LIN {X 0,Y 468.425,Z 168.39,A -85,B 0,C 180,E1 -7424.985,E2 -7424.985} C_VEL
LIN {X 0,Y 468.931,Z 154.374,A -85,B 0,C 180,E1 -7427.874,E2 -7427.874} C_VEL
LIN {X 0,Y 468.145,Z 148.139,A -85,B 0,C 180,E1 -7429.228,E2 -7429.228} C_VEL
LIN {X 0,Y 467.613,Z 145.238,A -85,B 0,C 180,E1 -7429.882,E2 -7429.882} C_VEL
LIN {X 0,Y 467.525,Z 145.248,A -85,B 0,C 180,E1 -7433.037,E2 -7433.037} C_VEL
LIN {X 0,Y 467.572,Z 145.242,A -85,B 0,C 180,E1 -7436.21,E2 -7436.21} C_VEL
LIN {X 0,Y 467.553,Z 145.24,A -85,B 0,C 180,E1 -7439.264,E2 -7439.264} C_VEL
LIN {X 0,Y 467.553,Z 145.247,A -85,B 0,C 180,E1 -7442.482,E2 -7442.482} C_VEL
LIN {X 0,Y 467.557,Z 145.24,A -85,B 0,C 180,E1 -7445.109,E2 -7445.109} C_VEL
LIN {X 0,Y 467.526,Z 145.247,A -85,B 0,C 180,E1 -7447.925,E2 -7447.925} C_VEL
LIN {X 0,Y 467.557,Z 145.242,A -85,B 0,C 180,E1 -7450.689,E2 -7450.689} C_VEL
LIN {X 0,Y 467.599,Z 145.243,A -85,B 0,C 180,E1 -7454.139,E2 -7454.139} C_VEL
LIN {X 0,Y 467.654,Z 145.23,A -85,B 0,C 180,E1 -7457.646,E2 -7457.646} C_VEL
LIN {X 0,Y 467.622,Z 145.234,A -85,B 0,C 180,E1 -7460.483,E2 -7460.483} C_VEL
LIN {X 0,Y 467.656,Z 145.227,A -85,B 0,C 180,E1 -7463.094,E2 -7463.094} C_VEL
LIN {X 0,Y 467.704,Z 145.221,A -85,B 0,C 180,E1 -7464.826,E2 -7464.826} C_VEL
LIN {X 0,Y 467.816,Z 145.21,A -85,B 0,C 180,E1 -7467.416,E2 -7467.416} C_VEL
LIN {X 0,Y 467.853,Z 145.208,A -85,B 0,C 180,E1 -7469.999,E2 -7469.999} C_VEL
LIN {X 0,Y 467.816,Z 145.207,A -85,B 0,C 180,E1 -7472.582,E2 -7472.582} C_VEL
LIN {X 0,Y 467.697,Z 145.226,A -85,B 0,C 180,E1 -7476.037,E2 -7476.037} C_VEL
LIN {X 0,Y 467.636,Z 145.23,A -85,B 0,C 180,E1 -7478.643,E2 -7478.643} C_VEL
LIN {X 0,Y 467.651,Z 145.228,A -85,B 0,C 180,E1 -7482.353,E2 -7482.353} C_VEL
LIN {X 0,Y 467.602,Z 145.237,A -85,B 0,C 180,E1 -7485.862,E2 -7485.862} C_VEL
LIN {X 0,Y 467.554,Z 145.247,A -85,B 0,C 180,E1 -7489.31,E2 -7489.31} C_VEL
LIN {X 0,Y 467.522,Z 145.244,A -85,B 0,C 180,E1 -7492.074,E2 -7492.074} C_VEL
LIN {X 0,Y 467.559,Z 145.242,A -85,B 0,C 180,E1 -7494.889,E2 -7494.889} C_VEL
LIN {X 0,Y 467.543,Z 145.243,A -85,B 0,C 180,E1 -7497.773,E2 -7497.773} C_VEL
LIN {X 0,Y 467.536,Z 145.249,A -85,B 0,C 180,E1 -7501.037,E2 -7501.037} C_VEL
LIN {X 0,Y 467.575,Z 145.237,A -85,B 0,C 180,E1 -7504.239,E2 -7504.239} C_VEL
LIN {X 0,Y 467.54,Z 145.248,A -85,B 0,C 180,E1 -7507.184,E2 -7507.184} C_VEL
LIN {X 0,Y 467.555,Z 145.24,A -85,B 0,C 180,E1 -7510.266,E2 -7510.266} C_VEL
LIN {X 0,Y 467.541,Z 145.242,A -85,B 0,C 180,E1 -7513.745,E2 -7513.745} C_VEL
LIN {X 0,Y 467.541,Z 145.243,A -85,B 0,C 180,E1 -7516.253,E2 -7516.253} C_VEL
LIN {X 0,Y 467.552,Z 145.24,A -85,B 0,C 180,E1 -7519.732,E2 -7519.732} C_VEL
LIN {X 0,Y 467.533,Z 145.249,A -85,B 0,C 180,E1 -7522.815,E2 -7522.815} C_VEL
LIN {X 0,Y 467.571,Z 145.238,A -85,B 0,C 180,E1 -7525.759,E2 -7525.759} C_VEL
LIN {X 0,Y 467.537,Z 145.245,A -85,B 0,C 180,E1 -7528.96,E2 -7528.96} C_VEL
LIN {X 0,Y 467.537,Z 145.246,A -85,B 0,C 180,E1 -7532.225,E2 -7532.225} C_VEL
LIN {X 0,Y 467.552,Z 145.241,A -85,B 0,C 180,E1 -7535.109,E2 -7535.109} C_VEL
LIN {X 0,Y 467.518,Z 145.247,A -85,B 0,C 180,E1 -7537.925,E2 -7537.925} C_VEL
LIN {X 0,Y 467.609,Z 145.237,A -85,B 0,C 180,E1 -7540.691,E2 -7540.691} C_VEL
LIN {X 0,Y 467.605,Z 145.241,A -85,B 0,C 180,E1 -7544.304,E2 -7544.304} C_VEL
LIN {X 0,Y 467.64,Z 145.233,A -85,B 0,C 180,E1 -7547.854,E2 -7547.854} C_VEL
LIN {X 0,Y 467.625,Z 145.231,A -85,B 0,C 180,E1 -7551.356,E2 -7551.356} C_VEL
LIN {X 0,Y 467.695,Z 145.229,A -85,B 0,C 180,E1 -7553.962,E2 -7553.962} C_VEL
LIN {X 0,Y 467.804,Z 145.21,A -85,B 0,C 180,E1 -7557.417,E2 -7557.417} C_VEL
LIN {X 0,Y 467.841,Z 145.212,A -85,B 0,C 180,E1 -7560,E2 -7560} C_VEL
LIN {X 0,Y 467.804,Z 145.209,A -85,B 0,C 180,E1 -7562.583,E2 -7562.583} C_VEL
LIN {X 0,Y 467.692,Z 145.228,A -85,B 0,C 180,E1 -7566.038,E2 -7566.038} C_VEL
LIN {X 0,Y 467.624,Z 145.231,A -85,B 0,C 180,E1 -7568.644,E2 -7568.644} C_VEL
LIN {X 0,Y 467.639,Z 145.232,A -85,B 0,C 180,E1 -7572.146,E2 -7572.146} C_VEL
LIN {X 0,Y 467.604,Z 145.241,A -85,B 0,C 180,E1 -7575.696,E2 -7575.696} C_VEL
LIN {X 0,Y 467.564,Z 145.239,A -85,B 0,C 180,E1 -7578.748,E2 -7578.748} C_VEL
LIN {X 0,Y 467.55,Z 145.245,A -85,B 0,C 180,E1 -7581.261,E2 -7581.261} C_VEL
LIN {X 0,Y 467.541,Z 145.244,A -85,B 0,C 180,E1 -7583.945,E2 -7583.945} C_VEL
LIN {X 0,Y 467.526,Z 145.245,A -85,B 0,C 180,E1 -7586.806,E2 -7586.806} C_VEL
LIN {X 0,Y 467.502,Z 145.249,A -85,B 0,C 180,E1 -7589.742,E2 -7589.742} C_VEL
LIN {X 0,Y 467.565,Z 145.241,A -85,B 0,C 180,E1 -7592.76,E2 -7592.76} C_VEL
LIN {X 0,Y 467.536,Z 145.243,A -85,B 0,C 180,E1 -7595.891,E2 -7595.891} C_VEL
LIN {X 0,Y 467.536,Z 145.25,A -85,B 0,C 180,E1 -7599.149,E2 -7599.149} C_VEL
LIN {X 0,Y 467.552,Z 145.244,A -85,B 0,C 180,E1 -7601.406,E2 -7601.406} C_VEL
LIN {X 0,Y 467.556,Z 145.247,A -85,B 0,C 180,E1 -7605.053,E2 -7605.053} C_VEL
LIN {X 0,Y 467.555,Z 145.245,A -85,B 0,C 180,E1 -7608.727,E2 -7608.727} C_VEL
LIN {X 0,Y 467.535,Z 145.242,A -85,B 0,C 180,E1 -7611.954,E2 -7611.954} C_VEL
LIN {X 0,Y 467.545,Z 145.244,A -85,B 0,C 180,E1 -7615.167,E2 -7615.167} C_VEL
LIN {X 0,Y 467.542,Z 145.244,A -85,B 0,C 180,E1 -7618.258,E2 -7618.258} C_VEL
LIN {X 0,Y 467.521,Z 145.247,A -85,B 0,C 180,E1 -7621.248,E2 -7621.248} C_VEL
LIN {X 0,Y 467.555,Z 145.345,A -85,B 0,C 180,E1 -7624.376,E2 -7624.376} C_VEL
LIN {X 0,Y 469.577,Z 155.706,A -85,B 0,C 180,E1 -7626.4,E2 -7626.4} C_VEL
LIN {X 0,Y 469.686,Z 160.79,A -85,B 0,C 180,E1 -7627.338,E2 -7627.338} C_VEL
LIN {X 0,Y 469.023,Z 174.71,A -85,B 0,C 180,E1 -7629.841,E2 -7629.841} C_VEL
LIN {X 0,Y 468.327,Z 192.765,A -85,B 0,C 180,E1 -7633.041,E2 -7633.041} C_VEL
LIN {X 0,Y 471.066,Z 211.841,A -85,B 0,C 180,E1 -7633.457,E2 -7633.457} C_VEL
LIN {X 0,Y 470.265,Z 300.839,A -85,B 0,C 180,E1 -7634.923,E2 -7634.923} C_VEL
LIN {X 0,Y 469.84,Z 314.649,A -85,B 0,C 180,E1 -7635.325,E2 -7635.325} C_VEL
LIN {X 0,Y 469.462,Z 327.139,A -85,B 0,C 180,E1 -7635.866,E2 -7635.866} C_VEL
LIN {X 0,Y 468.985,Z 339.105,A -85,B 0,C 180,E1 -7636.57,E2 -7636.57} C_VEL
LIN {X 0,Y 468.506,Z 350.327,A -85,B 0,C 180,E1 -7637.415,E2 -7637.415} C_VEL
LIN {X 0,Y 468.06,Z 360.974,A -85,B 0,C 180,E1 -7638.415,E2 -7638.415} C_VEL
LIN {X 0,Y 467.63,Z 369.45,A -85,B 0,C 180,E1 -7639.392,E2 -7639.392} C_VEL
LIN {X 0,Y 467.262,Z 378.639,A -85,B 0,C 180,E1 -7640.696,E2 -7640.696} C_VEL
LIN {X 0,Y 467.005,Z 386.039,A -85,B 0,C 180,E1 -7641.999,E2 -7641.999} C_VEL
LIN {X 0,Y 466.832,Z 391.044,A -85,B 0,C 180,E1 -7643.083,E2 -7643.083} C_VEL
LIN {X 0,Y 466.755,Z 395.897,A -85,B 0,C 180,E1 -7644.384,E2 -7644.384} C_VEL
LIN {X 0,Y 466.645,Z 399.603,A -85,B 0,C 180,E1 -7645.682,E2 -7645.682} C_VEL
LIN {X 0,Y 466.688,Z 401.518,A -85,B 0,C 180,E1 -7646.547,E2 -7646.547} C_VEL
LIN {X 0,Y 466.662,Z 402.961,A -85,B 0,C 180,E1 -7647.411,E2 -7647.411} C_VEL
LIN {X 0,Y 466.62,Z 404.599,A -85,B 0,C 180,E1 -7649.138,E2 -7649.138} C_VEL
LIN {X 0,Y 466.601,Z 404.823,A -85,B 0,C 180,E1 -7650.001,E2 -7650.001} C_VEL
LIN {X 0,Y 466.62,Z 404.604,A -85,B 0,C 180,E1 -7650.864,E2 -7650.864} C_VEL
LIN {X 0,Y 466.662,Z 402.957,A -85,B 0,C 180,E1 -7652.59,E2 -7652.59} C_VEL
LIN {X 0,Y 466.688,Z 401.525,A -85,B 0,C 180,E1 -7653.454,E2 -7653.454} C_VEL
LIN {X 0,Y 466.687,Z 398.517,A -85,B 0,C 180,E1 -7654.752,E2 -7654.752} C_VEL
LIN {X 0,Y 466.743,Z 394.447,A -85,B 0,C 180,E1 -7656.051,E2 -7656.051} C_VEL
LIN {X 0,Y 466.94,Z 388.181,A -85,B 0,C 180,E1 -7657.568,E2 -7657.568} C_VEL
LIN {X 0,Y 467.178,Z 381.351,A -85,B 0,C 180,E1 -7658.871,E2 -7658.871} C_VEL
LIN {X 0,Y 467.489,Z 372.873,A -85,B 0,C 180,E1 -7660.175,E2 -7660.175} C_VEL
LIN {X 0,Y 467.968,Z 364.14,A -85,B 0,C 180,E1 -7661.259,E2 -7661.259} C_VEL
LIN {X 0,Y 468.42,Z 354.024,A -85,B 0,C 180,E1 -7662.287,E2 -7662.287} C_VEL
LIN {X 0,Y 468.849,Z 342.723,A -85,B 0,C 180,E1 -7663.215,E2 -7663.215} C_VEL
LIN {X 0,Y 469.375,Z 330.864,A -85,B 0,C 180,E1 -7663.972,E2 -7663.972} C_VEL
LIN {X 0,Y 469.874,Z 317.322,A -85,B 0,C 180,E1 -7664.62,E2 -7664.62} C_VEL
LIN {X 0,Y 470.259,Z 305.288,A -85,B 0,C 180,E1 -7665.023,E2 -7665.023} C_VEL
LIN {X 0,Y 470.505,Z 290.619,A -85,B 0,C 180,E1 -7665.32,E2 -7665.32} C_VEL
LIN {X 0,Y 471.152,Z 209.638,A -85,B 0,C 180,E1 -7666.67,E2 -7666.67} C_VEL
LIN {X 0,Y 468.296,Z 191.81,A -85,B 0,C 180,E1 -7667.102,E2 -7667.102} C_VEL
LIN {X 0,Y 468.849,Z 176.842,A -85,B 0,C 180,E1 -7669.711,E2 -7669.711} C_VEL
LIN {X 0,Y 469.422,Z 162.683,A -85,B 0,C 180,E1 -7672.213,E2 -7672.213} C_VEL
LIN {X 0,Y 469.596,Z 156.216,A -85,B 0,C 180,E1 -7673.366,E2 -7673.366} C_VEL
LIN {X 0,Y 467.567,Z 145.248,A -85,B 0,C 180,E1 -7675.477,E2 -7675.477} C_VEL
LIN {X 0,Y 467.527,Z 145.25,A -85,B 0,C 180,E1 -7678.754,E2 -7678.754} C_VEL
LIN {X 0,Y 467.549,Z 145.246,A -85,B 0,C 180,E1 -7681.743,E2 -7681.743} C_VEL
LIN {X 0,Y 467.553,Z 145.246,A -85,B 0,C 180,E1 -7684.834,E2 -7684.834} C_VEL
LIN {X 0,Y 467.543,Z 145.243,A -85,B 0,C 180,E1 -7688.047,E2 -7688.047} C_VEL
LIN {X 0,Y 467.563,Z 145.243,A -85,B 0,C 180,E1 -7691.275,E2 -7691.275} C_VEL
LIN {X 0,Y 467.568,Z 145.243,A -85,B 0,C 180,E1 -7694.948,E2 -7694.948} C_VEL
LIN {X 0,Y 467.561,Z 145.242,A -85,B 0,C 180,E1 -7698.595,E2 -7698.595} C_VEL
LIN {X 0,Y 467.546,Z 145.24,A -85,B 0,C 180,E1 -7701.412,E2 -7701.412} C_VEL
LIN {X 0,Y 467.558,Z 145.242,A -85,B 0,C 180,E1 -7704.262,E2 -7704.262} C_VEL
LIN {X 0,Y 467.576,Z 145.239,A -85,B 0,C 180,E1 -7707.323,E2 -7707.323} C_VEL
LIN {X 0,Y 467.548,Z 145.245,A -85,B 0,C 180,E1 -7710.673,E2 -7710.673} C_VEL
LIN {X 0,Y 467.537,Z 145.243,A -85,B 0,C 180,E1 -7713.195,E2 -7713.195} C_VEL
LIN {X 0,Y 467.559,Z 145.245,A -85,B 0,C 180,E1 -7716.056,E2 -7716.056} C_VEL
LIN {X 0,Y 467.622,Z 145.233,A -85,B 0,C 180,E1 -7719.777,E2 -7719.777} C_VEL
LIN {X 0,Y 467.569,Z 145.243,A -85,B 0,C 180,E1 -7722.505,E2 -7722.505} C_VEL
LIN {X 0,Y 467.598,Z 145.237,A -85,B 0,C 180,E1 -7725.196,E2 -7725.196} C_VEL
LIN {X 0,Y 467.66,Z 145.234,A -85,B 0,C 180,E1 -7727.855,E2 -7727.855} C_VEL
LIN {X 0,Y 467.661,Z 145.232,A -85,B 0,C 180,E1 -7731.357,E2 -7731.357} C_VEL
LIN {X 0,Y 467.706,Z 145.23,A -85,B 0,C 180,E1 -7733.962,E2 -7733.962} C_VEL
LIN {X 0,Y 467.818,Z 145.214,A -85,B 0,C 180,E1 -7737.417,E2 -7737.417} C_VEL
LIN {X 0,Y 467.856,Z 145.211,A -85,B 0,C 180,E1 -7740,E2 -7740} C_VEL
LIN {X 0,Y 467.853,Z 145.209,A -85,B 0,C 180,E1 -7742.583,E2 -7742.583} C_VEL
LIN {X 0,Y 467.724,Z 145.348,A -85,B 0,C 180,E1 -7746.444,E2 -7746.444} C_VEL
LIN {X 0,Y 468.878,Z 151.823,A -85,B 0,C 180,E1 -7747.753,E2 -7747.753} C_VEL
LIN {X 0,Y 468.773,Z 162.022,A -85,B 0,C 180,E1 -7749.71,E2 -7749.71} C_VEL
LIN {X 0,Y 468.622,Z 168.72,A -85,B 0,C 180,E1 -7750.969,E2 -7750.969} C_VEL
LIN {X 0,Y 471.42,Z 183.099,A -85,B 0,C 180,E1 -7751.339,E2 -7751.339} C_VEL
LIN {X 0,Y 470.458,Z 276.646,A -85,B 0,C 180,E1 -7752.922,E2 -7752.922} C_VEL
LIN {X 0,Y 470.148,Z 290.015,A -85,B 0,C 180,E1 -7753.322,E2 -7753.322} C_VEL
LIN {X 0,Y 469.795,Z 303.075,A -85,B 0,C 180,E1 -7753.904,E2 -7753.904} C_VEL
LIN {X 0,Y 469.333,Z 315.18,A -85,B 0,C 180,E1 -7754.637,E2 -7754.637} C_VEL
LIN {X 0,Y 468.823,Z 326.843,A -85,B 0,C 180,E1 -7755.543,E2 -7755.543} C_VEL
LIN {X 0,Y 468.316,Z 337.266,A -85,B 0,C 180,E1 -7756.567,E2 -7756.567} C_VEL
LIN {X 0,Y 467.878,Z 346.668,A -85,B 0,C 180,E1 -7757.709,E2 -7757.709} C_VEL
LIN {X 0,Y 467.493,Z 355.126,A -85,B 0,C 180,E1 -7758.975,E2 -7758.975} C_VEL
LIN {X 0,Y 467.146,Z 361.925,A -85,B 0,C 180,E1 -7760.245,E2 -7760.245} C_VEL
LIN {X 0,Y 466.949,Z 367.849,A -85,B 0,C 180,E1 -7761.639,E2 -7761.639} C_VEL
LIN {X 0,Y 466.798,Z 372.451,A -85,B 0,C 180,E1 -7763.045,E2 -7763.045} C_VEL
LIN {X 0,Y 466.725,Z 374.852,A -85,B 0,C 180,E1 -7763.99,E2 -7763.99} C_VEL
LIN {X 0,Y 466.556,Z 377.331,A -85,B 0,C 180,E1 -7765.335,E2 -7765.335} C_VEL
LIN {X 0,Y 466.544,Z 378.893,A -85,B 0,C 180,E1 -7766.867,E2 -7766.867} C_VEL
LIN {X 0,Y 466.505,Z 379.236,A -85,B 0,C 180,E1 -7767.842,E2 -7767.842} C_VEL
LIN {X 0,Y 466.532,Z 378.9,A -85,B 0,C 180,E1 -7769.104,E2 -7769.104} C_VEL
LIN {X 0,Y 466.628,Z 377.107,A -85,B 0,C 180,E1 -7770.803,E2 -7770.803} C_VEL
LIN {X 0,Y 466.699,Z 375.248,A -85,B 0,C 180,E1 -7771.808,E2 -7771.808} C_VEL
LIN {X 0,Y 466.779,Z 371.323,A -85,B 0,C 180,E1 -7773.337,E2 -7773.337} C_VEL
LIN {X 0,Y 466.91,Z 367.439,A -85,B 0,C 180,E1 -7774.463,E2 -7774.463} C_VEL
LIN {X 0,Y 467.154,Z 361.069,A -85,B 0,C 180,E1 -7775.926,E2 -7775.926} C_VEL
LIN {X 0,Y 467.5,Z 353.312,A -85,B 0,C 180,E1 -7777.309,E2 -7777.309} C_VEL
LIN {X 0,Y 467.913,Z 343.957,A -85,B 0,C 180,E1 -7778.644,E2 -7778.644} C_VEL
LIN {X 0,Y 468.329,Z 334.292,A -85,B 0,C 180,E1 -7779.744,E2 -7779.744} C_VEL
LIN {X 0,Y 468.739,Z 323.844,A -85,B 0,C 180,E1 -7780.709,E2 -7780.709} C_VEL
LIN {X 0,Y 469.264,Z 311.997,A -85,B 0,C 180,E1 -7781.579,E2 -7781.579} C_VEL
LIN {X 0,Y 469.719,Z 299.794,A -85,B 0,C 180,E1 -7782.263,E2 -7782.263} C_VEL
LIN {X 0,Y 470.054,Z 286.143,A -85,B 0,C 180,E1 -7782.823,E2 -7782.823} C_VEL
LIN {X 0,Y 470.329,Z 272.94,A -85,B 0,C 180,E1 -7783.165,E2 -7783.165} C_VEL
LIN {X 0,Y 470.929,Z 213.093,A -85,B 0,C 180,E1 -7784.14,E2 -7784.14} C_VEL
LIN {X 0,Y 470.465,Z 207.289,A -85,B 0,C 180,E1 -7784.254,E2 -7784.254} C_VEL
LIN {X 0,Y 468.205,Z 197.882,A -85,B 0,C 180,E1 -7784.487,E2 -7784.487} C_VEL
LIN {X 0,Y 465.943,Z 190.424,A -85,B 0,C 180,E1 -7784.691,E2 -7784.691} C_VEL
LIN {X 0,Y 464.135,Z 182.84,A -85,B 0,C 180,E1 -7784.882,E2 -7784.882} C_VEL
LIN {X 0,Y 461.432,Z 168.53,A -85,B 0,C 180,E1 -7785.235,E2 -7785.235} C_VEL
LIN {X 0,Y 461.964,Z 155.386,A -85,B 0,C 180,E1 -7787.98,E2 -7787.98} C_VEL
LIN {X 0,Y 461.065,Z 148.726,A -85,B 0,C 180,E1 -7789.445,E2 -7789.445} C_VEL
LIN {X 0,Y 460.572,Z 146.116,A -85,B 0,C 180,E1 -7790.053,E2 -7790.053} C_VEL
LIN {X 0,Y 460.475,Z 146.124,A -85,B 0,C 180,E1 -7793.47,E2 -7793.47} C_VEL
LIN {X 0,Y 460.522,Z 146.122,A -85,B 0,C 180,E1 -7796.674,E2 -7796.674} C_VEL
LIN {X 0,Y 460.49,Z 146.121,A -85,B 0,C 180,E1 -7799.758,E2 -7799.758} C_VEL
LIN {X 0,Y 460.493,Z 146.123,A -85,B 0,C 180,E1 -7802.75,E2 -7802.75} C_VEL
LIN {X 0,Y 460.517,Z 146.117,A -85,B 0,C 180,E1 -7805.666,E2 -7805.666} C_VEL
LIN {X 0,Y 460.519,Z 146.12,A -85,B 0,C 180,E1 -7808.581,E2 -7808.581} C_VEL
LIN {X 0,Y 460.535,Z 146.114,A -85,B 0,C 180,E1 -7811.308,E2 -7811.308} C_VEL
LIN {X 0,Y 460.572,Z 146.117,A -85,B 0,C 180,E1 -7814.057,E2 -7814.057} C_VEL
LIN {X 0,Y 460.609,Z 146.108,A -85,B 0,C 180,E1 -7817.665,E2 -7817.665} C_VEL
LIN {X 0,Y 460.593,Z 146.107,A -85,B 0,C 180,E1 -7821.222,E2 -7821.222} C_VEL
LIN {X 0,Y 460.672,Z 146.105,A -85,B 0,C 180,E1 -7823.869,E2 -7823.869} C_VEL
LIN {X 0,Y 460.759,Z 146.088,A -85,B 0,C 180,E1 -7827.377,E2 -7827.377} C_VEL
LIN {X 0,Y 460.823,Z 146.084,A -85,B 0,C 180,E1 -7829.999,E2 -7829.999} C_VEL
LIN {X 0,Y 460.759,Z 146.086,A -85,B 0,C 180,E1 -7832.622,E2 -7832.622} C_VEL
LIN {X 0,Y 460.664,Z 146.101,A -85,B 0,C 180,E1 -7836.13,E2 -7836.13} C_VEL
LIN {X 0,Y 460.591,Z 146.107,A -85,B 0,C 180,E1 -7838.776,E2 -7838.776} C_VEL
LIN {X 0,Y 460.6,Z 146.106,A -85,B 0,C 180,E1 -7842.434,E2 -7842.434} C_VEL
LIN {X 0,Y 460.559,Z 146.113,A -85,B 0,C 180,E1 -7845.977,E2 -7845.977} C_VEL
LIN {X 0,Y 460.532,Z 146.116,A -85,B 0,C 180,E1 -7848.885,E2 -7848.885} C_VEL
LIN {X 0,Y 460.51,Z 146.124,A -85,B 0,C 180,E1 -7851.485,E2 -7851.485} C_VEL
LIN {X 0,Y 460.517,Z 146.116,A -85,B 0,C 180,E1 -7854.333,E2 -7854.333} C_VEL
LIN {X 0,Y 460.491,Z 146.128,A -85,B 0,C 180,E1 -7857.248,E2 -7857.248} C_VEL
LIN {X 0,Y 460.493,Z 146.12,A -85,B 0,C 180,E1 -7860.24,E2 -7860.24} C_VEL
LIN {X 0,Y 460.515,Z 146.122,A -85,B 0,C 180,E1 -7863.325,E2 -7863.325} C_VEL
LIN {X 0,Y 460.47,Z 146.124,A -85,B 0,C 180,E1 -7866.529,E2 -7866.529} C_VEL
LIN {X 0,Y 460.51,Z 146.117,A -85,B 0,C 180,E1 -7869.863,E2 -7869.863} C_VEL
LIN {X 0,Y 460.459,Z 146.132,A -85,B 0,C 180,E1 -7872.892,E2 -7872.892} C_VEL
LIN {X 0,Y 460.499,Z 146.119,A -85,B 0,C 180,E1 -7875.831,E2 -7875.831} C_VEL
LIN {X 0,Y 460.51,Z 146.123,A -85,B 0,C 180,E1 -7878.986,E2 -7878.986} C_VEL
LIN {X 0,Y 460.489,Z 146.124,A -85,B 0,C 180,E1 -7882.375,E2 -7882.375} C_VEL
LIN {X 0,Y 460.53,Z 146.115,A -85,B 0,C 180,E1 -7885.622,E2 -7885.622} C_VEL
LIN {X 0,Y 460.498,Z 146.125,A -85,B 0,C 180,E1 -7888.741,E2 -7888.741} C_VEL
LIN {X 0,Y 460.498,Z 146.119,A -85,B 0,C 180,E1 -7891.763,E2 -7891.763} C_VEL
LIN {X 0,Y 460.516,Z 146.122,A -85,B 0,C 180,E1 -7894.702,E2 -7894.702} C_VEL
LIN {X 0,Y 460.496,Z 146.119,A -85,B 0,C 180,E1 -7897.57,E2 -7897.57} C_VEL
LIN {X 0,Y 460.554,Z 146.12,A -85,B 0,C 180,E1 -7900.384,E2 -7900.384} C_VEL
LIN {X 0,Y 460.56,Z 146.116,A -85,B 0,C 180,E1 -7904.057,E2 -7904.057} C_VEL
LIN {X 0,Y 460.596,Z 146.108,A -85,B 0,C 180,E1 -7907.665,E2 -7907.665} C_VEL
LIN {X 0,Y 460.58,Z 146.109,A -85,B 0,C 180,E1 -7911.223,E2 -7911.223} C_VEL
LIN {X 0,Y 460.661,Z 146.104,A -85,B 0,C 180,E1 -7913.869,E2 -7913.869} C_VEL
LIN {X 0,Y 460.748,Z 146.089,A -85,B 0,C 180,E1 -7917.377,E2 -7917.377} C_VEL
LIN {X 0,Y 460.811,Z 146.087,A -85,B 0,C 180,E1 -7920,E2 -7920} C_VEL
LIN {X 0,Y 460.747,Z 146.088,A -85,B 0,C 180,E1 -7922.623,E2 -7922.623} C_VEL
LIN {X 0,Y 460.658,Z 146.103,A -85,B 0,C 180,E1 -7926.13,E2 -7926.13} C_VEL
LIN {X 0,Y 460.579,Z 146.109,A -85,B 0,C 180,E1 -7928.777,E2 -7928.777} C_VEL
LIN {X 0,Y 460.589,Z 146.108,A -85,B 0,C 180,E1 -7932.435,E2 -7932.435} C_VEL
LIN {X 0,Y 460.549,Z 146.116,A -85,B 0,C 180,E1 -7935.978,E2 -7935.978} C_VEL
LIN {X 0,Y 460.522,Z 146.117,A -85,B 0,C 180,E1 -7938.887,E2 -7938.887} C_VEL
LIN {X 0,Y 460.501,Z 146.127,A -85,B 0,C 180,E1 -7941.486,E2 -7941.486} C_VEL
LIN {X 0,Y 460.505,Z 146.118,A -85,B 0,C 180,E1 -7944.334,E2 -7944.334} C_VEL
LIN {X 0,Y 460.481,Z 146.127,A -85,B 0,C 180,E1 -7947.25,E2 -7947.25} C_VEL
LIN {X 0,Y 460.471,Z 146.122,A -85,B 0,C 180,E1 -7950.243,E2 -7950.243} C_VEL
LIN {X 0,Y 460.508,Z 146.125,A -85,B 0,C 180,E1 -7953.327,E2 -7953.327} C_VEL
LIN {X 0,Y 460.453,Z 146.125,A -85,B 0,C 180,E1 -7956.532,E2 -7956.532} C_VEL
LIN {X 0,Y 460.503,Z 146.119,A -85,B 0,C 180,E1 -7959.865,E2 -7959.865} C_VEL
LIN {X 0,Y 460.45,Z 146.131,A -85,B 0,C 180,E1 -7962.893,E2 -7962.893} C_VEL
LIN {X 0,Y 460.498,Z 146.119,A -85,B 0,C 180,E1 -7965.832,E2 -7965.832} C_VEL
LIN {X 0,Y 460.509,Z 146.125,A -85,B 0,C 180,E1 -7968.988,E2 -7968.988} C_VEL
LIN {X 0,Y 460.478,Z 146.124,A -85,B 0,C 180,E1 -7972.376,E2 -7972.376} C_VEL
LIN {X 0,Y 460.529,Z 146.115,A -85,B 0,C 180,E1 -7975.623,E2 -7975.623} C_VEL
LIN {X 0,Y 460.501,Z 146.127,A -85,B 0,C 180,E1 -7978.743,E2 -7978.743} C_VEL
LIN {X 0,Y 460.493,Z 146.121,A -85,B 0,C 180,E1 -7981.764,E2 -7981.764} C_VEL
LIN {X 0,Y 460.544,Z 146.127,A -85,B 0,C 180,E1 -7984.16,E2 -7984.16} C_VEL
LIN {X 0,Y 462.734,Z 157.978,A -85,B 0,C 180,E1 -7986.505,E2 -7986.505} C_VEL
LIN {X 0,Y 462.406,Z 169.387,A -85,B 0,C 180,E1 -7988.607,E2 -7988.607} C_VEL
LIN {X 0,Y 461.565,Z 185.829,A -85,B 0,C 180,E1 -7991.583,E2 -7991.583} C_VEL
LIN {X 0,Y 461.332,Z 192.537,A -85,B 0,C 180,E1 -7992.79,E2 -7992.79} C_VEL
LIN {X 0,Y 464.237,Z 212.61,A -85,B 0,C 180,E1 -7993.238,E2 -7993.238} C_VEL
LIN {X 0,Y 463.352,Z 301.882,A -85,B 0,C 180,E1 -7994.749,E2 -7994.749} C_VEL
LIN {X 0,Y 462.91,Z 315.28,A -85,B 0,C 180,E1 -7995.156,E2 -7995.156} C_VEL
LIN {X 0,Y 462.495,Z 327.522,A -85,B 0,C 180,E1 -7995.705,E2 -7995.705} C_VEL
LIN {X 0,Y 461.97,Z 340.146,A -85,B 0,C 180,E1 -7996.474,E2 -7996.474} C_VEL
LIN {X 0,Y 461.451,Z 351.822,A -85,B 0,C 180,E1 -7997.389,E2 -7997.389} C_VEL
LIN {X 0,Y 461.005,Z 361.575,A -85,B 0,C 180,E1 -7998.347,E2 -7998.347} C_VEL
LIN {X 0,Y 460.515,Z 370.744,A -85,B 0,C 180,E1 -7999.448,E2 -7999.448} C_VEL
LIN {X 0,Y 460.173,Z 379.692,A -85,B 0,C 180,E1 -8000.773,E2 -8000.773} C_VEL
LIN {X 0,Y 459.887,Z 386.845,A -85,B 0,C 180,E1 -8002.095,E2 -8002.095} C_VEL
LIN {X 0,Y 459.713,Z 393.112,A -85,B 0,C 180,E1 -8003.57,E2 -8003.57} C_VEL
LIN {X 0,Y 459.614,Z 398.275,A -85,B 0,C 180,E1 -8005.176,E2 -8005.176} C_VEL
LIN {X 0,Y 459.583,Z 401.294,A -85,B 0,C 180,E1 -8006.494,E2 -8006.494} C_VEL
LIN {X 0,Y 459.584,Z 402.749,A -85,B 0,C 180,E1 -8007.371,E2 -8007.371} C_VEL
LIN {X 0,Y 459.523,Z 404.397,A -85,B 0,C 180,E1 -8009.124,E2 -8009.124} C_VEL
LIN {X 0,Y 459.532,Z 404.627,A -85,B 0,C 180,E1 -8010.001,E2 -8010.001} C_VEL
LIN {X 0,Y 459.523,Z 404.413,A -85,B 0,C 180,E1 -8010.877,E2 -8010.877} C_VEL
LIN {X 0,Y 459.584,Z 402.77,A -85,B 0,C 180,E1 -8012.63,E2 -8012.63} C_VEL
LIN {X 0,Y 459.583,Z 401.339,A -85,B 0,C 180,E1 -8013.508,E2 -8013.508} C_VEL
LIN {X 0,Y 459.615,Z 398.334,A -85,B 0,C 180,E1 -8014.825,E2 -8014.825} C_VEL
LIN {X 0,Y 459.693,Z 393.3,A -85,B 0,C 180,E1 -8016.407,E2 -8016.407} C_VEL
LIN {X 0,Y 459.891,Z 386.977,A -85,B 0,C 180,E1 -8017.906,E2 -8017.906} C_VEL
LIN {X 0,Y 460.177,Z 379.912,A -85,B 0,C 180,E1 -8019.229,E2 -8019.229} C_VEL
LIN {X 0,Y 460.534,Z 371.052,A -85,B 0,C 180,E1 -8020.553,E2 -8020.553} C_VEL
LIN {X 0,Y 461.1,Z 361.007,A -85,B 0,C 180,E1 -8021.763,E2 -8021.763} C_VEL
LIN {X 0,Y 461.561,Z 350.198,A -85,B 0,C 180,E1 -8022.807,E2 -8022.807} C_VEL
LIN {X 0,Y 462.082,Z 339.476,A -85,B 0,C 180,E1 -8023.636,E2 -8023.636} C_VEL
LIN {X 0,Y 462.65,Z 326.791,A -85,B 0,C 180,E1 -8024.404,E2 -8024.404} C_VEL
LIN {X 0,Y 463.144,Z 313.719,A -85,B 0,C 180,E1 -8024.978,E2 -8024.978} C_VEL
LIN {X 0,Y 463.549,Z 300.995,A -85,B 0,C 180,E1 -8025.359,E2 -8025.359} C_VEL
LIN {X 0,Y 464.427,Z 210.669,A -85,B 0,C 180,E1 -8026.92,E2 -8026.92} C_VEL
LIN {X 0,Y 461.386,Z 191.495,A -85,B 0,C 180,E1 -8027.407,E2 -8027.407} C_VEL
LIN {X 0,Y 461.973,Z 175.505,A -85,B 0,C 180,E1 -8030.249,E2 -8030.249} C_VEL
LIN {X 0,Y 462.713,Z 160.018,A -85,B 0,C 180,E1 -8033.024,E2 -8033.024} C_VEL
LIN {X 0,Y 462.253,Z 154.911,A -85,B 0,C 180,E1 -8033.989,E2 -8033.989} C_VEL
LIN {X 0,Y 460.533,Z 146.124,A -85,B 0,C 180,E1 -8035.736,E2 -8035.736} C_VEL
LIN {X 0,Y 460.498,Z 146.124,A -85,B 0,C 180,E1 -8038.237,E2 -8038.237} C_VEL
LIN {X 0,Y 460.498,Z 146.126,A -85,B 0,C 180,E1 -8041.278,E2 -8041.278} C_VEL
LIN {X 0,Y 460.522,Z 146.119,A -85,B 0,C 180,E1 -8044.503,E2 -8044.503} C_VEL
LIN {X 0,Y 460.486,Z 146.124,A -85,B 0,C 180,E1 -8047.625,E2 -8047.625} C_VEL
LIN {X 0,Y 460.517,Z 146.123,A -85,B 0,C 180,E1 -8051.014,E2 -8051.014} C_VEL
LIN {X 0,Y 460.514,Z 146.121,A -85,B 0,C 180,E1 -8054.59,E2 -8054.59} C_VEL
LIN {X 0,Y 460.477,Z 146.12,A -85,B 0,C 180,E1 -8057.813,E2 -8057.813} C_VEL
LIN {X 0,Y 460.513,Z 146.118,A -85,B 0,C 180,E1 -8060.136,E2 -8060.136} C_VEL
LIN {X 0,Y 460.473,Z 146.121,A -85,B 0,C 180,E1 -8063.47,E2 -8063.47} C_VEL
LIN {X 0,Y 460.519,Z 146.121,A -85,B 0,C 180,E1 -8066.674,E2 -8066.674} C_VEL
LIN {X 0,Y 460.5,Z 146.119,A -85,B 0,C 180,E1 -8069.759,E2 -8069.759} C_VEL
LIN {X 0,Y 460.493,Z 146.123,A -85,B 0,C 180,E1 -8072.751,E2 -8072.751} C_VEL
LIN {X 0,Y 460.521,Z 146.118,A -85,B 0,C 180,E1 -8075.667,E2 -8075.667} C_VEL
LIN {X 0,Y 460.525,Z 146.117,A -85,B 0,C 180,E1 -8078.579,E2 -8078.579} C_VEL
LIN {X 0,Y 460.586,Z 146.109,A -85,B 0,C 180,E1 -8081.311,E2 -8081.311} C_VEL
LIN {X 0,Y 460.554,Z 146.114,A -85,B 0,C 180,E1 -8084.965,E2 -8084.965} C_VEL
LIN {X 0,Y 460.613,Z 146.109,A -85,B 0,C 180,E1 -8088.559,E2 -8088.559} C_VEL
LIN {X 0,Y 460.613,Z 146.109,A -85,B 0,C 180,E1 -8091.224,E2 -8091.224} C_VEL
LIN {X 0,Y 460.672,Z 146.105,A -85,B 0,C 180,E1 -8093.87,E2 -8093.87} C_VEL
LIN {X 0,Y 460.761,Z 146.092,A -85,B 0,C 180,E1 -8097.377,E2 -8097.377} C_VEL
LIN {X 0,Y 460.826,Z 146.087,A -85,B 0,C 180,E1 -8100,E2 -8100} C_VEL
LIN {X 0,Y 460.793,Z 146.088,A -85,B 0,C 180,E1 -8102.623,E2 -8102.623} C_VEL
LIN {X 0,Y 460.687,Z 146.11,A -85,B 0,C 180,E1 -8106.185,E2 -8106.185} C_VEL
LIN {X 0,Y 461.968,Z 153.202,A -85,B 0,C 180,E1 -8107.65,E2 -8107.65} C_VEL
LIN {X 0,Y 461.842,Z 163.447,A -85,B 0,C 180,E1 -8109.636,E2 -8109.636} C_VEL
LIN {X 0,Y 461.679,Z 168.768,A -85,B 0,C 180,E1 -8110.664,E2 -8110.664} C_VEL
LIN {X 0,Y 464.739,Z 184.49,A -85,B 0,C 180,E1 -8111.09,E2 -8111.09} C_VEL
LIN {X 0,Y 463.599,Z 277.445,A -85,B 0,C 180,E1 -8112.698,E2 -8112.698} C_VEL
LIN {X 0,Y 463.27,Z 291.145,A -85,B 0,C 180,E1 -8113.126,E2 -8113.126} C_VEL
LIN {X 0,Y 462.943,Z 303.362,A -85,B 0,C 180,E1 -8113.688,E2 -8113.688} C_VEL
LIN {X 0,Y 462.473,Z 315.133,A -85,B 0,C 180,E1 -8114.409,E2 -8114.409} C_VEL
LIN {X 0,Y 461.927,Z 326.852,A -85,B 0,C 180,E1 -8115.329,E2 -8115.329} C_VEL
LIN {X 0,Y 461.38,Z 336.985,A -85,B 0,C 180,E1 -8116.33,E2 -8116.33} C_VEL
LIN {X 0,Y 460.902,Z 346.749,A -85,B 0,C 180,E1 -8117.527,E2 -8117.527} C_VEL
LIN {X 0,Y 460.496,Z 354.502,A -85,B 0,C 180,E1 -8118.693,E2 -8118.693} C_VEL
LIN {X 0,Y 460.2,Z 360.897,A -85,B 0,C 180,E1 -8119.865,E2 -8119.865} C_VEL
LIN {X 0,Y 459.935,Z 366.947,A -85,B 0,C 180,E1 -8121.233,E2 -8121.233} C_VEL
LIN {X 0,Y 459.761,Z 371.239,A -85,B 0,C 180,E1 -8122.468,E2 -8122.468} C_VEL
LIN {X 0,Y 459.646,Z 375.022,A -85,B 0,C 180,E1 -8123.903,E2 -8123.903} C_VEL
LIN {X 0,Y 459.452,Z 377.823,A -85,B 0,C 180,E1 -8125.511,E2 -8125.511} C_VEL
LIN {X 0,Y 459.433,Z 378.72,A -85,B 0,C 180,E1 -8126.335,E2 -8126.335} C_VEL
LIN {X 0,Y 459.428,Z 379.372,A -85,B 0,C 180,E1 -8127.47,E2 -8127.47} C_VEL
LIN {X 0,Y 459.421,Z 379.403,A -85,B 0,C 180,E1 -8128.309,E2 -8128.309} C_VEL
LIN {X 0,Y 459.452,Z 378.973,A -85,B 0,C 180,E1 -8129.319,E2 -8129.319} C_VEL
LIN {X 0,Y 459.5,Z 377.992,A -85,B 0,C 180,E1 -8130.314,E2 -8130.314} C_VEL
LIN {X 0,Y 459.612,Z 375.457,A -85,B 0,C 180,E1 -8131.84,E2 -8131.84} C_VEL
LIN {X 0,Y 459.705,Z 371.533,A -85,B 0,C 180,E1 -8133.393,E2 -8133.393} C_VEL
LIN {X 0,Y 459.902,Z 365.977,A -85,B 0,C 180,E1 -8134.964,E2 -8134.964} C_VEL
LIN {X 0,Y 460.18,Z 360.314,A -85,B 0,C 180,E1 -8136.209,E2 -8136.209} C_VEL
LIN {X 0,Y 460.56,Z 352.317,A -85,B 0,C 180,E1 -8137.618,E2 -8137.618} C_VEL
LIN {X 0,Y 460.958,Z 343.247,A -85,B 0,C 180,E1 -8138.893,E2 -8138.893} C_VEL
LIN {X 0,Y 461.371,Z 333.3,A -85,B 0,C 180,E1 -8140.019,E2 -8140.019} C_VEL
LIN {X 0,Y 461.863,Z 322.415,A -85,B 0,C 180,E1 -8141.013,E2 -8141.013} C_VEL
LIN {X 0,Y 462.415,Z 310.487,A -85,B 0,C 180,E1 -8141.864,E2 -8141.864} C_VEL
LIN {X 0,Y 462.853,Z 298.815,A -85,B 0,C 180,E1 -8142.508,E2 -8142.508} C_VEL
LIN {X 0,Y 463.161,Z 285.506,A -85,B 0,C 180,E1 -8143.047,E2 -8143.047} C_VEL
LIN {X 0,Y 463.454,Z 271.899,A -85,B 0,C 180,E1 -8143.392,E2 -8143.392} C_VEL
LIN {X 0,Y 464.368,Z 184.32,A -85,B 0,C 180,E1 -8144.849,E2 -8144.849} C_VEL
LIN {X 0,Y 464.135,Z 182.84,A -85,B 0,C 180,E1 -8144.882,E2 -8144.882} C_VEL
LIN {X 0,Y 462.835,Z 178.939,A -85,B 0,C 180,E1 -8144.998,E2 -8144.998} C_VEL
LIN {X 0,Y 458.955,Z 173.288,A -85,B 0,C 180,E1 -8145.234,E2 -8145.234} C_VEL
LIN {X 0,Y 455.978,Z 169.433,A -85,B 0,C 180,E1 -8145.543,E2 -8145.543} C_VEL
LIN {X 0,Y 454.674,Z 166.881,A -85,B 0,C 180,E1 -8145.884,E2 -8145.884} C_VEL
LIN {X 0,Y 454.587,Z 166.153,A -85,B 0,C 180,E1 -8146.021,E2 -8146.021} C_VEL
LIN {X 0,Y 454.945,Z 155.075,A -85,B 0,C 180,E1 -8148.373,E2 -8148.373} C_VEL
LIN {X 0,Y 453.499,Z 146.997,A -85,B 0,C 180,E1 -8150.226,E2 -8150.226} C_VEL
LIN {X 0,Y 453.453,Z 146.999,A -85,B 0,C 180,E1 -8153.702,E2 -8153.702} C_VEL
LIN {X 0,Y 453.486,Z 146.996,A -85,B 0,C 180,E1 -8156.813,E2 -8156.813} C_VEL
LIN {X 0,Y 453.452,Z 147.002,A -85,B 0,C 180,E1 -8160.266,E2 -8160.266} C_VEL
LIN {X 0,Y 453.431,Z 146.999,A -85,B 0,C 180,E1 -8163.288,E2 -8163.288} C_VEL
LIN {X 0,Y 453.485,Z 147,A -85,B 0,C 180,E1 -8166.237,E2 -8166.237} C_VEL
LIN {X 0,Y 453.465,Z 146.995,A -85,B 0,C 180,E1 -8169.116,E2 -8169.116} C_VEL
LIN {X 0,Y 453.465,Z 147,A -85,B 0,C 180,E1 -8171.942,E2 -8171.942} C_VEL
LIN {X 0,Y 453.52,Z 146.989,A -85,B 0,C 180,E1 -8174.725,E2 -8174.725} C_VEL
LIN {X 0,Y 453.55,Z 146.988,A -85,B 0,C 180,E1 -8178.378,E2 -8178.378} C_VEL
LIN {X 0,Y 453.563,Z 146.983,A -85,B 0,C 180,E1 -8181.085,E2 -8181.085} C_VEL
LIN {X 0,Y 453.64,Z 146.979,A -85,B 0,C 180,E1 -8183.773,E2 -8183.773} C_VEL
LIN {X 0,Y 453.706,Z 146.967,A -85,B 0,C 180,E1 -8187.336,E2 -8187.336} C_VEL
LIN {X 0,Y 453.772,Z 146.962,A -85,B 0,C 180,E1 -8189.999,E2 -8189.999} C_VEL
LIN {X 0,Y 453.706,Z 146.965,A -85,B 0,C 180,E1 -8192.663,E2 -8192.663} C_VEL
LIN {X 0,Y 453.632,Z 146.976,A -85,B 0,C 180,E1 -8196.225,E2 -8196.225} C_VEL
LIN {X 0,Y 453.561,Z 146.984,A -85,B 0,C 180,E1 -8198.913,E2 -8198.913} C_VEL
LIN {X 0,Y 453.567,Z 146.982,A -85,B 0,C 180,E1 -8202.528,E2 -8202.528} C_VEL
LIN {X 0,Y 453.499,Z 146.991,A -85,B 0,C 180,E1 -8206.197,E2 -8206.197} C_VEL
LIN {X 0,Y 453.487,Z 146.995,A -85,B 0,C 180,E1 -8209.026,E2 -8209.026} C_VEL
LIN {X 0,Y 453.472,Z 146.996,A -85,B 0,C 180,E1 -8211.835,E2 -8211.835} C_VEL
LIN {X 0,Y 453.469,Z 146.996,A -85,B 0,C 180,E1 -8214.736,E2 -8214.736} C_VEL
LIN {X 0,Y 453.461,Z 146.996,A -85,B 0,C 180,E1 -8217.941,E2 -8217.941} C_VEL
LIN {X 0,Y 453.452,Z 146.999,A -85,B 0,C 180,E1 -8220.76,E2 -8220.76} C_VEL
LIN {X 0,Y 453.465,Z 146.995,A -85,B 0,C 180,E1 -8223.913,E2 -8223.913} C_VEL
LIN {X 0,Y 453.447,Z 147.003,A -85,B 0,C 180,E1 -8227.189,E2 -8227.189} C_VEL
LIN {X 0,Y 453.467,Z 146.998,A -85,B 0,C 180,E1 -8230.611,E2 -8230.611} C_VEL
LIN {X 0,Y 453.478,Z 146.997,A -85,B 0,C 180,E1 -8234.527,E2 -8234.527} C_VEL
LIN {X 0,Y 453.432,Z 147,A -85,B 0,C 180,E1 -8238.07,E2 -8238.07} C_VEL
LIN {X 0,Y 453.436,Z 147.006,A -85,B 0,C 180,E1 -8240.801,E2 -8240.801} C_VEL
LIN {X 0,Y 453.444,Z 146.998,A -85,B 0,C 180,E1 -8243.916,E2 -8243.916} C_VEL
LIN {X 0,Y 453.468,Z 146.996,A -85,B 0,C 180,E1 -8247.15,E2 -8247.15} C_VEL
LIN {X 0,Y 453.45,Z 147.001,A -85,B 0,C 180,E1 -8250.266,E2 -8250.266} C_VEL
LIN {X 0,Y 453.435,Z 146.999,A -85,B 0,C 180,E1 -8253.289,E2 -8253.289} C_VEL
LIN {X 0,Y 453.485,Z 146.998,A -85,B 0,C 180,E1 -8256.237,E2 -8256.237} C_VEL
LIN {X 0,Y 453.467,Z 146.995,A -85,B 0,C 180,E1 -8259.117,E2 -8259.117} C_VEL
LIN {X 0,Y 453.477,Z 146.997,A -85,B 0,C 180,E1 -8261.943,E2 -8261.943} C_VEL
LIN {X 0,Y 453.511,Z 146.992,A -85,B 0,C 180,E1 -8264.725,E2 -8264.725} C_VEL
LIN {X 0,Y 453.537,Z 146.991,A -85,B 0,C 180,E1 -8268.378,E2 -8268.378} C_VEL
LIN {X 0,Y 453.55,Z 146.984,A -85,B 0,C 180,E1 -8271.086,E2 -8271.086} C_VEL
LIN {X 0,Y 453.629,Z 146.979,A -85,B 0,C 180,E1 -8273.774,E2 -8273.774} C_VEL
LIN {X 0,Y 453.694,Z 146.967,A -85,B 0,C 180,E1 -8277.336,E2 -8277.336} C_VEL
LIN {X 0,Y 453.78,Z 146.963,A -85,B 0,C 180,E1 -8280,E2 -8280} C_VEL
LIN {X 0,Y 453.694,Z 146.967,A -85,B 0,C 180,E1 -8282.663,E2 -8282.663} C_VEL
LIN {X 0,Y 453.626,Z 146.978,A -85,B 0,C 180,E1 -8286.226,E2 -8286.226} C_VEL
LIN {X 0,Y 453.549,Z 146.985,A -85,B 0,C 180,E1 -8288.914,E2 -8288.914} C_VEL
LIN {X 0,Y 453.557,Z 146.984,A -85,B 0,C 180,E1 -8292.529,E2 -8292.529} C_VEL
LIN {X 0,Y 453.488,Z 146.993,A -85,B 0,C 180,E1 -8296.198,E2 -8296.198} C_VEL
LIN {X 0,Y 453.477,Z 146.995,A -85,B 0,C 180,E1 -8299.028,E2 -8299.028} C_VEL
LIN {X 0,Y 453.461,Z 146.999,A -85,B 0,C 180,E1 -8301.837,E2 -8301.837} C_VEL
LIN {X 0,Y 453.459,Z 146.996,A -85,B 0,C 180,E1 -8304.738,E2 -8304.738} C_VEL
LIN {X 0,Y 453.449,Z 146.998,A -85,B 0,C 180,E1 -8307.942,E2 -8307.942} C_VEL
LIN {X 0,Y 453.439,Z 147,A -85,B 0,C 180,E1 -8310.762,E2 -8310.762} C_VEL
LIN {X 0,Y 453.458,Z 146.997,A -85,B 0,C 180,E1 -8313.914,E2 -8313.914} C_VEL
LIN {X 0,Y 453.429,Z 147.007,A -85,B 0,C 180,E1 -8317.192,E2 -8317.192} C_VEL
LIN {X 0,Y 453.463,Z 146.997,A -85,B 0,C 180,E1 -8320.612,E2 -8320.612} C_VEL
LIN {X 0,Y 453.475,Z 146.996,A -85,B 0,C 180,E1 -8324.529,E2 -8324.529} C_VEL
LIN {X 0,Y 453.429,Z 147,A -85,B 0,C 180,E1 -8328.072,E2 -8328.072} C_VEL
LIN {X 0,Y 453.433,Z 147.006,A -85,B 0,C 180,E1 -8330.803,E2 -8330.803} C_VEL
LIN {X 0,Y 453.437,Z 146.999,A -85,B 0,C 180,E1 -8333.917,E2 -8333.917} C_VEL
LIN {X 0,Y 453.467,Z 146.998,A -85,B 0,C 180,E1 -8337.151,E2 -8337.151} C_VEL
LIN {X 0,Y 453.443,Z 147.002,A -85,B 0,C 180,E1 -8340.267,E2 -8340.267} C_VEL
LIN {X 0,Y 453.436,Z 147.004,A -85,B 0,C 180,E1 -8343.29,E2 -8343.29} C_VEL
LIN {X 0,Y 453.488,Z 147.099,A -85,B 0,C 180,E1 -8343.977,E2 -8343.977} C_VEL
LIN {X 0,Y 455.739,Z 158.964,A -85,B 0,C 180,E1 -8346.363,E2 -8346.363} C_VEL
LIN {X 0,Y 455.446,Z 170.378,A -85,B 0,C 180,E1 -8348.502,E2 -8348.502} C_VEL
LIN {X 0,Y 454.55,Z 186.811,A -85,B 0,C 180,E1 -8351.522,E2 -8351.522} C_VEL
LIN {X 0,Y 454.375,Z 192.592,A -85,B 0,C 180,E1 -8352.545,E2 -8352.545} C_VEL
LIN {X 0,Y 457.392,Z 212.344,A -85,B 0,C 180,E1 -8353,E2 -8353} C_VEL
LIN {X 0,Y 456.459,Z 300.62,A -85,B 0,C 180,E1 -8354.513,E2 -8354.513} C_VEL
LIN {X 0,Y 456.028,Z 314.352,A -85,B 0,C 180,E1 -8354.927,E2 -8354.927} C_VEL
LIN {X 0,Y 455.565,Z 326.809,A -85,B 0,C 180,E1 -8355.483,E2 -8355.483} C_VEL
LIN {X 0,Y 455.089,Z 337.972,A -85,B 0,C 180,E1 -8356.152,E2 -8356.152} C_VEL
LIN {X 0,Y 454.541,Z 350.117,A -85,B 0,C 180,E1 -8357.089,E2 -8357.089} C_VEL
LIN {X 0,Y 454.016,Z 361.145,A -85,B 0,C 180,E1 -8358.165,E2 -8358.165} C_VEL
LIN {X 0,Y 453.501,Z 370.357,A -85,B 0,C 180,E1 -8359.283,E2 -8359.283} C_VEL
LIN {X 0,Y 453.114,Z 379.342,A -85,B 0,C 180,E1 -8360.628,E2 -8360.628} C_VEL
LIN {X 0,Y 452.836,Z 386.54,A -85,B 0,C 180,E1 -8361.971,E2 -8361.971} C_VEL
LIN {X 0,Y 452.609,Z 393.335,A -85,B 0,C 180,E1 -8363.605,E2 -8363.605} C_VEL
LIN {X 0,Y 452.542,Z 398.025,A -85,B 0,C 180,E1 -8365.101,E2 -8365.101} C_VEL
LIN {X 0,Y 452.48,Z 401.06,A -85,B 0,C 180,E1 -8366.439,E2 -8366.439} C_VEL
LIN {X 0,Y 452.507,Z 402.532,A -85,B 0,C 180,E1 -8367.33,E2 -8367.33} C_VEL
LIN {X 0,Y 452.429,Z 404.193,A -85,B 0,C 180,E1 -8369.111,E2 -8369.111} C_VEL
LIN {X 0,Y 452.437,Z 404.429,A -85,B 0,C 180,E1 -8370.001,E2 -8370.001} C_VEL
LIN {X 0,Y 452.429,Z 404.224,A -85,B 0,C 180,E1 -8370.891,E2 -8370.891} C_VEL
LIN {X 0,Y 452.508,Z 402.587,A -85,B 0,C 180,E1 -8372.671,E2 -8372.671} C_VEL
LIN {X 0,Y 452.479,Z 401.16,A -85,B 0,C 180,E1 -8373.563,E2 -8373.563} C_VEL
LIN {X 0,Y 452.543,Z 398.157,A -85,B 0,C 180,E1 -8374.901,E2 -8374.901} C_VEL
LIN {X 0,Y 452.611,Z 393.54,A -85,B 0,C 180,E1 -8376.397,E2 -8376.397} C_VEL
LIN {X 0,Y 452.805,Z 387.841,A -85,B 0,C 180,E1 -8377.806,E2 -8377.806} C_VEL
LIN {X 0,Y 453.066,Z 381.017,A -85,B 0,C 180,E1 -8379.15,E2 -8379.15} C_VEL
LIN {X 0,Y 453.438,Z 372.55,A -85,B 0,C 180,E1 -8380.494,E2 -8380.494} C_VEL
LIN {X 0,Y 453.958,Z 363.834,A -85,B 0,C 180,E1 -8381.611,E2 -8381.611} C_VEL
LIN {X 0,Y 454.536,Z 352.832,A -85,B 0,C 180,E1 -8382.755,E2 -8382.755} C_VEL
LIN {X 0,Y 455.004,Z 342.488,A -85,B 0,C 180,E1 -8383.625,E2 -8383.625} C_VEL
LIN {X 0,Y 455.613,Z 330.736,A -85,B 0,C 180,E1 -8384.403,E2 -8384.403} C_VEL
LIN {X 0,Y 456.156,Z 317.318,A -85,B 0,C 180,E1 -8385.07,E2 -8385.07} C_VEL
LIN {X 0,Y 456.613,Z 304.57,A -85,B 0,C 180,E1 -8385.512,E2 -8385.512} C_VEL
LIN {X 0,Y 456.907,Z 289.882,A -85,B 0,C 180,E1 -8385.816,E2 -8385.816} C_VEL
LIN {X 0,Y 457.71,Z 211.751,A -85,B 0,C 180,E1 -8387.177,E2 -8387.177} C_VEL
LIN {X 0,Y 454.45,Z 191.34,A -85,B 0,C 180,E1 -8387.703,E2 -8387.703} C_VEL
LIN {X 0,Y 455.016,Z 176.739,A -85,B 0,C 180,E1 -8390.337,E2 -8390.337} C_VEL
LIN {X 0,Y 455.768,Z 162.584,A -85,B 0,C 180,E1 -8392.915,E2 -8392.915} C_VEL
LIN {X 0,Y 455.723,Z 158.724,A -85,B 0,C 180,E1 -8393.639,E2 -8393.639} C_VEL
LIN {X 0,Y 453.763,Z 148.405,A -85,B 0,C 180,E1 -8395.702,E2 -8395.702} C_VEL
LIN {X 0,Y 453.46,Z 147.005,A -85,B 0,C 180,E1 -8396.014,E2 -8396.014} C_VEL
LIN {X 0,Y 453.45,Z 147.004,A -85,B 0,C 180,E1 -8398.717,E2 -8398.717} C_VEL
LIN {X 0,Y 453.444,Z 147.003,A -85,B 0,C 180,E1 -8401.802,E2 -8401.802} C_VEL
LIN {X 0,Y 453.475,Z 147.002,A -85,B 0,C 180,E1 -8404.99,E2 -8404.99} C_VEL
LIN {X 0,Y 453.448,Z 147,A -85,B 0,C 180,E1 -8408.314,E2 -8408.314} C_VEL
LIN {X 0,Y 453.473,Z 146.999,A -85,B 0,C 180,E1 -8410.612,E2 -8410.612} C_VEL
LIN {X 0,Y 453.484,Z 146.996,A -85,B 0,C 180,E1 -8414.529,E2 -8414.529} C_VEL
LIN {X 0,Y 453.438,Z 146.998,A -85,B 0,C 180,E1 -8418.071,E2 -8418.071} C_VEL
LIN {X 0,Y 453.443,Z 147,A -85,B 0,C 180,E1 -8420.802,E2 -8420.802} C_VEL
LIN {X 0,Y 453.452,Z 146.997,A -85,B 0,C 180,E1 -8423.917,E2 -8423.917} C_VEL
LIN {X 0,Y 453.477,Z 146.996,A -85,B 0,C 180,E1 -8427.151,E2 -8427.151} C_VEL
LIN {X 0,Y 453.459,Z 147,A -85,B 0,C 180,E1 -8430.267,E2 -8430.267} C_VEL
LIN {X 0,Y 453.444,Z 146.998,A -85,B 0,C 180,E1 -8433.29,E2 -8433.29} C_VEL
LIN {X 0,Y 453.496,Z 146.996,A -85,B 0,C 180,E1 -8436.238,E2 -8436.238} C_VEL
LIN {X 0,Y 453.484,Z 146.991,A -85,B 0,C 180,E1 -8439.118,E2 -8439.118} C_VEL
LIN {X 0,Y 453.489,Z 146.996,A -85,B 0,C 180,E1 -8441.944,E2 -8441.944} C_VEL
LIN {X 0,Y 453.524,Z 146.991,A -85,B 0,C 180,E1 -8444.726,E2 -8444.726} C_VEL
LIN {X 0,Y 453.562,Z 146.989,A -85,B 0,C 180,E1 -8448.379,E2 -8448.379} C_VEL
LIN {X 0,Y 453.581,Z 146.985,A -85,B 0,C 180,E1 -8451.087,E2 -8451.087} C_VEL
LIN {X 0,Y 453.64,Z 146.981,A -85,B 0,C 180,E1 -8453.774,E2 -8453.774} C_VEL
LIN {X 0,Y 453.708,Z 146.971,A -85,B 0,C 180,E1 -8457.337,E2 -8457.337} C_VEL
LIN {X 0,Y 453.795,Z 146.963,A -85,B 0,C 180,E1 -8460,E2 -8460} C_VEL
LIN {X 0,Y 453.737,Z 146.968,A -85,B 0,C 180,E1 -8462.664,E2 -8462.664} C_VEL
LIN {X 0,Y 453.662,Z 147.055,A -85,B 0,C 180,E1 -8465.947,E2 -8465.947} C_VEL
LIN {X 0,Y 455.069,Z 154.642,A -85,B 0,C 180,E1 -8467.543,E2 -8467.543} C_VEL
LIN {X 0,Y 454.92,Z 164.888,A -85,B 0,C 180,E1 -8469.56,E2 -8469.56} C_VEL
LIN {X 0,Y 454.828,Z 169.28,A -85,B 0,C 180,E1 -8470.377,E2 -8470.377} C_VEL
LIN {X 0,Y 458.036,Z 185.321,A -85,B 0,C 180,E1 -8470.819,E2 -8470.819} C_VEL
LIN {X 0,Y 456.816,Z 277.145,A -85,B 0,C 180,E1 -8472.438,E2 -8472.438} C_VEL
LIN {X 0,Y 456.497,Z 290.213,A -85,B 0,C 180,E1 -8472.843,E2 -8472.843} C_VEL
LIN {X 0,Y 456.112,Z 301.852,A -85,B 0,C 180,E1 -8473.364,E2 -8473.364} C_VEL
LIN {X 0,Y 455.663,Z 314.172,A -85,B 0,C 180,E1 -8474.106,E2 -8474.106} C_VEL
LIN {X 0,Y 455.059,Z 325.574,A -85,B 0,C 180,E1 -8474.993,E2 -8474.993} C_VEL
LIN {X 0,Y 454.501,Z 336.367,A -85,B 0,C 180,E1 -8476.046,E2 -8476.046} C_VEL
LIN {X 0,Y 454.049,Z 345.118,A -85,B 0,C 180,E1 -8477.103,E2 -8477.103} C_VEL
LIN {X 0,Y 453.591,Z 353.178,A -85,B 0,C 180,E1 -8478.286,E2 -8478.286} C_VEL
LIN {X 0,Y 453.185,Z 361.034,A -85,B 0,C 180,E1 -8479.713,E2 -8479.713} C_VEL
LIN {X 0,Y 452.937,Z 366.317,A -85,B 0,C 180,E1 -8480.909,E2 -8480.909} C_VEL
LIN {X 0,Y 452.701,Z 371.4,A -85,B 0,C 180,E1 -8482.356,E2 -8482.356} C_VEL
LIN {X 0,Y 452.574,Z 375.197,A -85,B 0,C 180,E1 -8483.813,E2 -8483.813} C_VEL
LIN {X 0,Y 452.426,Z 377.054,A -85,B 0,C 180,E1 -8484.798,E2 -8484.798} C_VEL
LIN {X 0,Y 452.346,Z 378.437,A -85,B 0,C 180,E1 -8485.788,E2 -8485.788} C_VEL
LIN {X 0,Y 452.322,Z 379.278,A -85,B 0,C 180,E1 -8486.782,E2 -8486.782} C_VEL
LIN {X 0,Y 452.319,Z 379.625,A -85,B 0,C 180,E1 -8487.784,E2 -8487.784} C_VEL
LIN {X 0,Y 452.322,Z 379.467,A -85,B 0,C 180,E1 -8488.795,E2 -8488.795} C_VEL
LIN {X 0,Y 452.388,Z 378.746,A -85,B 0,C 180,E1 -8489.811,E2 -8489.811} C_VEL
LIN {X 0,Y 452.494,Z 376.713,A -85,B 0,C 180,E1 -8491.323,E2 -8491.323} C_VEL
LIN {X 0,Y 452.58,Z 372.976,A -85,B 0,C 180,E1 -8493.012,E2 -8493.012} C_VEL
LIN {X 0,Y 452.782,Z 367.717,A -85,B 0,C 180,E1 -8494.647,E2 -8494.647} C_VEL
LIN {X 0,Y 453.05,Z 361.467,A -85,B 0,C 180,E1 -8496.121,E2 -8496.121} C_VEL
LIN {X 0,Y 453.439,Z 354.022,A -85,B 0,C 180,E1 -8497.494,E2 -8497.494} C_VEL
LIN {X 0,Y 453.865,Z 344.942,A -85,B 0,C 180,E1 -8498.839,E2 -8498.839} C_VEL
LIN {X 0,Y 454.304,Z 335.753,A -85,B 0,C 180,E1 -8499.941,E2 -8499.941} C_VEL
LIN {X 0,Y 454.808,Z 324.497,A -85,B 0,C 180,E1 -8501.023,E2 -8501.023} C_VEL
LIN {X 0,Y 455.333,Z 313.976,A -85,B 0,C 180,E1 -8501.832,E2 -8501.832} C_VEL
LIN {X 0,Y 455.831,Z 301.682,A -85,B 0,C 180,E1 -8502.571,E2 -8502.571} C_VEL
LIN {X 0,Y 456.209,Z 288.616,A -85,B 0,C 180,E1 -8503.146,E2 -8503.146} C_VEL
LIN {X 0,Y 456.476,Z 275.659,A -85,B 0,C 180,E1 -8503.531,E2 -8503.531} C_VEL
LIN {X 0,Y 457.504,Z 184.775,A -85,B 0,C 180,E1 -8505.086,E2 -8505.086} C_VEL
LIN {X 0,Y 454.485,Z 168.685,A -85,B 0,C 180,E1 -8505.491,E2 -8505.491} C_VEL
LIN {X 0,Y 454.587,Z 166.153,A -85,B 0,C 180,E1 -8506.021,E2 -8506.021} C_VEL
LIN {X 0,Y 454.085,Z 163.227,A -85,B 0,C 180,E1 -8506.666,E2 -8506.666} C_VEL
LIN {X 0,Y 451.407,Z 158.798,A -85,B 0,C 180,E1 -8507.737,E2 -8507.737} C_VEL
LIN {X 0,Y 447.845,Z 153.567,A -85,B 0,C 180,E1 -8509.047,E2 -8509.047} C_VEL
LIN {X 0,Y 447.194,Z 151.688,A -85,B 0,C 180,E1 -8509.492,E2 -8509.492} C_VEL
LIN {X 0,Y 446.442,Z 147.876,A -85,B 0,C 180,E1 -8510.426,E2 -8510.426} C_VEL
LIN {X 0,Y 446.406,Z 147.877,A -85,B 0,C 180,E1 -8513.411,E2 -8513.411} C_VEL
LIN {X 0,Y 446.455,Z 147.875,A -85,B 0,C 180,E1 -8516.566,E2 -8516.566} C_VEL
LIN {X 0,Y 446.419,Z 147.875,A -85,B 0,C 180,E1 -8519.983,E2 -8519.983} C_VEL
LIN {X 0,Y 446.39,Z 147.879,A -85,B 0,C 180,E1 -8522.833,E2 -8522.833} C_VEL
LIN {X 0,Y 446.424,Z 147.875,A -85,B 0,C 180,E1 -8525.937,E2 -8525.937} C_VEL
LIN {X 0,Y 446.446,Z 147.871,A -85,B 0,C 180,E1 -8528.772,E2 -8528.772} C_VEL
LIN {X 0,Y 446.417,Z 147.875,A -85,B 0,C 180,E1 -8531.647,E2 -8531.647} C_VEL
LIN {X 0,Y 446.46,Z 147.871,A -85,B 0,C 180,E1 -8534.477,E2 -8534.477} C_VEL
LIN {X 0,Y 446.522,Z 147.861,A -85,B 0,C 180,E1 -8537.384,E2 -8537.384} C_VEL
LIN {X 0,Y 446.514,Z 147.861,A -85,B 0,C 180,E1 -8540.943,E2 -8540.943} C_VEL
LIN {X 0,Y 446.61,Z 147.853,A -85,B 0,C 180,E1 -8543.675,E2 -8543.675} C_VEL
LIN {X 0,Y 446.655,Z 147.845,A -85,B 0,C 180,E1 -8547.294,E2 -8547.294} C_VEL
LIN {X 0,Y 446.722,Z 147.84,A -85,B 0,C 180,E1 -8549.999,E2 -8549.999} C_VEL
LIN {X 0,Y 446.656,Z 147.843,A -85,B 0,C 180,E1 -8552.705,E2 -8552.705} C_VEL
LIN {X 0,Y 446.603,Z 147.851,A -85,B 0,C 180,E1 -8556.324,E2 -8556.324} C_VEL
LIN {X 0,Y 446.512,Z 147.863,A -85,B 0,C 180,E1 -8559.055,E2 -8559.055} C_VEL
LIN {X 0,Y 446.524,Z 147.86,A -85,B 0,C 180,E1 -8562.729,E2 -8562.729} C_VEL
LIN {X 0,Y 446.452,Z 147.869,A -85,B 0,C 180,E1 -8566.206,E2 -8566.206} C_VEL
LIN {X 0,Y 446.433,Z 147.878,A -85,B 0,C 180,E1 -8569.304,E2 -8569.304} C_VEL
LIN {X 0,Y 446.413,Z 147.874,A -85,B 0,C 180,E1 -8572.199,E2 -8572.199} C_VEL
LIN {X 0,Y 446.421,Z 147.879,A -85,B 0,C 180,E1 -8575.153,E2 -8575.153} C_VEL
LIN {X 0,Y 446.416,Z 147.873,A -85,B 0,C 180,E1 -8578.182,E2 -8578.182} C_VEL
LIN {X 0,Y 446.392,Z 147.882,A -85,B 0,C 180,E1 -8581.301,E2 -8581.301} C_VEL
LIN {X 0,Y 446.42,Z 147.874,A -85,B 0,C 180,E1 -8584.523,E2 -8584.523} C_VEL
LIN {X 0,Y 446.408,Z 147.874,A -85,B 0,C 180,E1 -8588.077,E2 -8588.077} C_VEL
LIN {X 0,Y 446.397,Z 147.878,A -85,B 0,C 180,E1 -8591.393,E2 -8591.393} C_VEL
LIN {X 0,Y 446.446,Z 147.874,A -85,B 0,C 180,E1 -8595.103,E2 -8595.103} C_VEL
LIN {X 0,Y 446.396,Z 147.881,A -85,B 0,C 180,E1 -8598.605,E2 -8598.605} C_VEL
LIN {X 0,Y 446.4,Z 147.875,A -85,B 0,C 180,E1 -8601.922,E2 -8601.922} C_VEL
LIN {X 0,Y 446.416,Z 147.873,A -85,B 0,C 180,E1 -8605.475,E2 -8605.475} C_VEL
LIN {X 0,Y 446.402,Z 147.881,A -85,B 0,C 180,E1 -8608.698,E2 -8608.698} C_VEL
LIN {X 0,Y 446.418,Z 147.874,A -85,B 0,C 180,E1 -8611.836,E2 -8611.836} C_VEL
LIN {X 0,Y 446.415,Z 147.876,A -85,B 0,C 180,E1 -8614.845,E2 -8614.845} C_VEL
LIN {X 0,Y 446.44,Z 147.876,A -85,B 0,C 180,E1 -8618.245,E2 -8618.245} C_VEL
LIN {X 0,Y 446.432,Z 147.872,A -85,B 0,C 180,E1 -8621.648,E2 -8621.648} C_VEL
LIN {X 0,Y 446.451,Z 147.874,A -85,B 0,C 180,E1 -8624.477,E2 -8624.477} C_VEL
LIN {X 0,Y 446.509,Z 147.862,A -85,B 0,C 180,E1 -8627.384,E2 -8627.384} C_VEL
LIN {X 0,Y 446.501,Z 147.863,A -85,B 0,C 180,E1 -8630.944,E2 -8630.944} C_VEL
LIN {X 0,Y 446.599,Z 147.853,A -85,B 0,C 180,E1 -8633.675,E2 -8633.675} C_VEL
LIN {X 0,Y 446.644,Z 147.845,A -85,B 0,C 180,E1 -8637.294,E2 -8637.294} C_VEL
LIN {X 0,Y 446.729,Z 147.841,A -85,B 0,C 180,E1 -8640,E2 -8640} C_VEL
LIN {X 0,Y 446.644,Z 147.845,A -85,B 0,C 180,E1 -8642.705,E2 -8642.705} C_VEL
LIN {X 0,Y 446.596,Z 147.853,A -85,B 0,C 180,E1 -8646.324,E2 -8646.324} C_VEL
LIN {X 0,Y 446.5,Z 147.863,A -85,B 0,C 180,E1 -8649.056,E2 -8649.056} C_VEL
LIN {X 0,Y 446.513,Z 147.861,A -85,B 0,C 180,E1 -8652.73,E2 -8652.73} C_VEL
LIN {X 0,Y 446.442,Z 147.871,A -85,B 0,C 180,E1 -8656.207,E2 -8656.207} C_VEL
LIN {X 0,Y 446.423,Z 147.877,A -85,B 0,C 180,E1 -8659.305,E2 -8659.305} C_VEL
LIN {X 0,Y 446.399,Z 147.876,A -85,B 0,C 180,E1 -8662.201,E2 -8662.201} C_VEL
LIN {X 0,Y 446.412,Z 147.878,A -85,B 0,C 180,E1 -8665.155,E2 -8665.155} C_VEL
LIN {X 0,Y 446.407,Z 147.874,A -85,B 0,C 180,E1 -8668.184,E2 -8668.184} C_VEL
LIN {X 0,Y 446.384,Z 147.885,A -85,B 0,C 180,E1 -8671.303,E2 -8671.303} C_VEL
LIN {X 0,Y 446.413,Z 147.874,A -85,B 0,C 180,E1 -8674.524,E2 -8674.524} C_VEL
LIN {X 0,Y 446.391,Z 147.876,A -85,B 0,C 180,E1 -8678.077,E2 -8678.077} C_VEL
LIN {X 0,Y 446.393,Z 147.88,A -85,B 0,C 180,E1 -8681.395,E2 -8681.395} C_VEL
LIN {X 0,Y 446.443,Z 147.876,A -85,B 0,C 180,E1 -8685.105,E2 -8685.105} C_VEL
LIN {X 0,Y 446.394,Z 147.879,A -85,B 0,C 180,E1 -8688.606,E2 -8688.606} C_VEL
LIN {X 0,Y 446.392,Z 147.876,A -85,B 0,C 180,E1 -8691.925,E2 -8691.925} C_VEL
LIN {X 0,Y 446.415,Z 147.874,A -85,B 0,C 180,E1 -8695.477,E2 -8695.477} C_VEL
LIN {X 0,Y 446.387,Z 147.884,A -85,B 0,C 180,E1 -8698.698,E2 -8698.698} C_VEL
LIN {X 0,Y 446.398,Z 147.877,A -85,B 0,C 180,E1 -8701.843,E2 -8701.843} C_VEL
LIN {X 0,Y 446.434,Z 147.953,A -85,B 0,C 180,E1 -8703.765,E2 -8703.765} C_VEL
LIN {X 0,Y 448.741,Z 159.924,A -85,B 0,C 180,E1 -8706.217,E2 -8706.217} C_VEL
LIN {X 0,Y 448.568,Z 168.81,A -85,B 0,C 180,E1 -8707.913,E2 -8707.913} C_VEL
LIN {X 0,Y 447.631,Z 186.523,A -85,B 0,C 180,E1 -8711.226,E2 -8711.226} C_VEL
LIN {X 0,Y 447.413,Z 192.37,A -85,B 0,C 180,E1 -8712.285,E2 -8712.285} C_VEL
LIN {X 0,Y 450.541,Z 213.783,A -85,B 0,C 180,E1 -8712.784,E2 -8712.784} C_VEL
LIN {X 0,Y 449.555,Z 301.415,A -85,B 0,C 180,E1 -8714.327,E2 -8714.327} C_VEL
LIN {X 0,Y 449.101,Z 314.815,A -85,B 0,C 180,E1 -8714.747,E2 -8714.747} C_VEL
LIN {X 0,Y 448.614,Z 327.076,A -85,B 0,C 180,E1 -8715.311,E2 -8715.311} C_VEL
LIN {X 0,Y 448.089,Z 338.924,A -85,B 0,C 180,E1 -8716.047,E2 -8716.047} C_VEL
LIN {X 0,Y 447.53,Z 350.636,A -85,B 0,C 180,E1 -8716.978,E2 -8716.978} C_VEL
LIN {X 0,Y 447.048,Z 360.688,A -85,B 0,C 180,E1 -8717.978,E2 -8717.978} C_VEL
LIN {X 0,Y 446.504,Z 369.954,A -85,B 0,C 180,E1 -8719.113,E2 -8719.113} C_VEL
LIN {X 0,Y 446.057,Z 378.98,A -85,B 0,C 180,E1 -8720.478,E2 -8720.478} C_VEL
LIN {X 0,Y 445.764,Z 386.226,A -85,B 0,C 180,E1 -8721.843,E2 -8721.843} C_VEL
LIN {X 0,Y 445.553,Z 392.148,A -85,B 0,C 180,E1 -8723.252,E2 -8723.252} C_VEL
LIN {X 0,Y 445.474,Z 396.505,A -85,B 0,C 180,E1 -8724.569,E2 -8724.569} C_VEL
LIN {X 0,Y 445.41,Z 398.884,A -85,B 0,C 180,E1 -8725.476,E2 -8725.476} C_VEL
LIN {X 0,Y 445.378,Z 400.823,A -85,B 0,C 180,E1 -8726.382,E2 -8726.382} C_VEL
LIN {X 0,Y 445.432,Z 402.313,A -85,B 0,C 180,E1 -8727.288,E2 -8727.288} C_VEL
LIN {X 0,Y 445.339,Z 403.988,A -85,B 0,C 180,E1 -8729.097,E2 -8729.097} C_VEL
LIN {X 0,Y 445.344,Z 404.23,A -85,B 0,C 180,E1 -8730.001,E2 -8730.001} C_VEL
LIN {X 0,Y 445.339,Z 404.036,A -85,B 0,C 180,E1 -8730.905,E2 -8730.905} C_VEL
LIN {X 0,Y 445.433,Z 402.408,A -85,B 0,C 180,E1 -8732.714,E2 -8732.714} C_VEL
LIN {X 0,Y 445.377,Z 400.986,A -85,B 0,C 180,E1 -8733.62,E2 -8733.62} C_VEL
LIN {X 0,Y 445.471,Z 397.99,A -85,B 0,C 180,E1 -8734.979,E2 -8734.979} C_VEL
LIN {X 0,Y 445.53,Z 393.782,A -85,B 0,C 180,E1 -8736.386,E2 -8736.386} C_VEL
LIN {X 0,Y 445.726,Z 387.689,A -85,B 0,C 180,E1 -8737.931,E2 -8737.931} C_VEL
LIN {X 0,Y 446.042,Z 380.871,A -85,B 0,C 180,E1 -8739.295,E2 -8739.295} C_VEL
LIN {X 0,Y 446.433,Z 372.421,A -85,B 0,C 180,E1 -8740.66,E2 -8740.66} C_VEL
LIN {X 0,Y 446.98,Z 363.73,A -85,B 0,C 180,E1 -8741.795,E2 -8741.795} C_VEL
LIN {X 0,Y 447.554,Z 353.58,A -85,B 0,C 180,E1 -8742.877,E2 -8742.877} C_VEL
LIN {X 0,Y 448.107,Z 342.433,A -85,B 0,C 180,E1 -8743.839,E2 -8743.839} C_VEL
LIN {X 0,Y 448.729,Z 330.741,A -85,B 0,C 180,E1 -8744.629,E2 -8744.629} C_VEL
LIN {X 0,Y 449.326,Z 317.419,A -85,B 0,C 180,E1 -8745.305,E2 -8745.305} C_VEL
LIN {X 0,Y 449.79,Z 304.898,A -85,B 0,C 180,E1 -8745.753,E2 -8745.753} C_VEL
LIN {X 0,Y 450.112,Z 290.673,A -85,B 0,C 180,E1 -8746.062,E2 -8746.062} C_VEL
LIN {X 0,Y 450.979,Z 212.598,A -85,B 0,C 180,E1 -8747.452,E2 -8747.452} C_VEL
LIN {X 0,Y 447.498,Z 191.013,A -85,B 0,C 180,E1 -8748.041,E2 -8748.041} C_VEL
LIN {X 0,Y 448.142,Z 176.721,A -85,B 0,C 180,E1 -8750.663,E2 -8750.663} C_VEL
LIN {X 0,Y 448.923,Z 162.588,A -85,B 0,C 180,E1 -8753.285,E2 -8753.285} C_VEL
LIN {X 0,Y 448.297,Z 156.956,A -85,B 0,C 180,E1 -8754.391,E2 -8754.391} C_VEL
LIN {X 0,Y 446.392,Z 147.885,A -85,B 0,C 180,E1 -8756.299,E2 -8756.299} C_VEL
LIN {X 0,Y 446.41,Z 147.881,A -85,B 0,C 180,E1 -8759.213,E2 -8759.213} C_VEL
LIN {X 0,Y 446.41,Z 147.878,A -85,B 0,C 180,E1 -8762.363,E2 -8762.363} C_VEL
LIN {X 0,Y 446.424,Z 147.88,A -85,B 0,C 180,E1 -8765.052,E2 -8765.052} C_VEL
LIN {X 0,Y 446.4,Z 147.877,A -85,B 0,C 180,E1 -8768.077,E2 -8768.077} C_VEL
LIN {X 0,Y 446.403,Z 147.878,A -85,B 0,C 180,E1 -8771.395,E2 -8771.395} C_VEL
LIN {X 0,Y 446.452,Z 147.871,A -85,B 0,C 180,E1 -8775.104,E2 -8775.104} C_VEL
LIN {X 0,Y 446.403,Z 147.876,A -85,B 0,C 180,E1 -8778.606,E2 -8778.606} C_VEL
LIN {X 0,Y 446.407,Z 147.873,A -85,B 0,C 180,E1 -8781.923,E2 -8781.923} C_VEL
LIN {X 0,Y 446.424,Z 147.874,A -85,B 0,C 180,E1 -8785.477,E2 -8785.477} C_VEL
LIN {X 0,Y 446.411,Z 147.877,A -85,B 0,C 180,E1 -8788.699,E2 -8788.699} C_VEL
LIN {X 0,Y 446.427,Z 147.873,A -85,B 0,C 180,E1 -8791.837,E2 -8791.837} C_VEL
LIN {X 0,Y 446.425,Z 147.874,A -85,B 0,C 180,E1 -8794.846,E2 -8794.846} C_VEL
LIN {X 0,Y 446.452,Z 147.875,A -85,B 0,C 180,E1 -8798.246,E2 -8798.246} C_VEL
LIN {X 0,Y 446.443,Z 147.873,A -85,B 0,C 180,E1 -8801.649,E2 -8801.649} C_VEL
LIN {X 0,Y 446.464,Z 147.872,A -85,B 0,C 180,E1 -8804.478,E2 -8804.478} C_VEL
LIN {X 0,Y 446.52,Z 147.864,A -85,B 0,C 180,E1 -8807.384,E2 -8807.384} C_VEL
LIN {X 0,Y 446.529,Z 147.863,A -85,B 0,C 180,E1 -8810.945,E2 -8810.945} C_VEL
LIN {X 0,Y 446.61,Z 147.856,A -85,B 0,C 180,E1 -8813.676,E2 -8813.676} C_VEL
LIN {X 0,Y 446.658,Z 147.849,A -85,B 0,C 180,E1 -8817.295,E2 -8817.295} C_VEL
LIN {X 0,Y 446.765,Z 147.839,A -85,B 0,C 180,E1 -8820,E2 -8820} C_VEL
LIN {X 0,Y 446.684,Z 147.847,A -85,B 0,C 180,E1 -8822.706,E2 -8822.706} C_VEL
LIN {X 0,Y 446.634,Z 148.052,A -85,B 0,C 180,E1 -8825.701,E2 -8825.701} C_VEL
LIN {X 0,Y 448.247,Z 157.218,A -85,B 0,C 180,E1 -8827.659,E2 -8827.659} C_VEL
LIN {X 0,Y 447.893,Z 169.245,A -85,B 0,C 180,E1 -8830.052,E2 -8830.052} C_VEL
LIN {X 0,Y 451.312,Z 186.268,A -85,B 0,C 180,E1 -8830.536,E2 -8830.536} C_VEL
LIN {X 0,Y 450.046,Z 277.001,A -85,B 0,C 180,E1 -8832.171,E2 -8832.171} C_VEL
LIN {X 0,Y 449.693,Z 290.177,A -85,B 0,C 180,E1 -8832.581,E2 -8832.581} C_VEL
LIN {X 0,Y 449.267,Z 302.977,A -85,B 0,C 180,E1 -8833.168,E2 -8833.168} C_VEL
LIN {X 0,Y 448.822,Z 314.267,A -85,B 0,C 180,E1 -8833.867,E2 -8833.867} C_VEL
LIN {X 0,Y 448.192,Z 325.631,A -85,B 0,C 180,E1 -8834.763,E2 -8834.763} C_VEL
LIN {X 0,Y 447.577,Z 336.475,A -85,B 0,C 180,E1 -8835.833,E2 -8835.833} C_VEL
LIN {X 0,Y 447.086,Z 345.252,A -85,B 0,C 180,E1 -8836.906,E2 -8836.906} C_VEL
LIN {X 0,Y 446.61,Z 353.319,A -85,B 0,C 180,E1 -8838.107,E2 -8838.107} C_VEL
LIN {X 0,Y 446.166,Z 361.186,A -85,B 0,C 180,E1 -8839.556,E2 -8839.556} C_VEL
LIN {X 0,Y 445.883,Z 366.482,A -85,B 0,C 180,E1 -8840.772,E2 -8840.772} C_VEL
LIN {X 0,Y 445.636,Z 371.571,A -85,B 0,C 180,E1 -8842.241,E2 -8842.241} C_VEL
LIN {X 0,Y 445.497,Z 375.528,A -85,B 0,C 180,E1 -8843.795,E2 -8843.795} C_VEL
LIN {X 0,Y 445.305,Z 378.003,A -85,B 0,C 180,E1 -8845.222,E2 -8845.222} C_VEL
LIN {X 0,Y 445.234,Z 379.103,A -85,B 0,C 180,E1 -8846.231,E2 -8846.231} C_VEL
LIN {X 0,Y 445.234,Z 379.841,A -85,B 0,C 180,E1 -8847.875,E2 -8847.875} C_VEL
LIN {X 0,Y 445.299,Z 378.988,A -85,B 0,C 180,E1 -8849.767,E2 -8849.767} C_VEL
LIN {X 0,Y 445.417,Z 376.545,A -85,B 0,C 180,E1 -8851.565,E2 -8851.565} C_VEL
LIN {X 0,Y 445.52,Z 372.591,A -85,B 0,C 180,E1 -8853.272,E2 -8853.272} C_VEL
LIN {X 0,Y 445.739,Z 367.181,A -85,B 0,C 180,E1 -8854.925,E2 -8854.925} C_VEL
LIN {X 0,Y 446.037,Z 361.177,A -85,B 0,C 180,E1 -8856.317,E2 -8856.317} C_VEL
LIN {X 0,Y 446.399,Z 354.321,A -85,B 0,C 180,E1 -8857.595,E2 -8857.595} C_VEL
LIN {X 0,Y 446.861,Z 345.088,A -85,B 0,C 180,E1 -8858.984,E2 -8858.984} C_VEL
LIN {X 0,Y 447.318,Z 335.872,A -85,B 0,C 180,E1 -8860.104,E2 -8860.104} C_VEL
LIN {X 0,Y 447.788,Z 325.572,A -85,B 0,C 180,E1 -8861.117,E2 -8861.117} C_VEL
LIN {X 0,Y 448.433,Z 313.425,A -85,B 0,C 180,E1 -8862.067,E2 -8862.067} C_VEL
LIN {X 0,Y 448.922,Z 301.471,A -85,B 0,C 180,E1 -8862.786,E2 -8862.786} C_VEL
LIN {X 0,Y 449.323,Z 287.886,A -85,B 0,C 180,E1 -8863.384,E2 -8863.384} C_VEL
LIN {X 0,Y 449.609,Z 275.134,A -85,B 0,C 180,E1 -8863.757,E2 -8863.757} C_VEL
LIN {X 0,Y 450.677,Z 185.652,A -85,B 0,C 180,E1 -8865.313,E2 -8865.313} C_VEL
LIN {X 0,Y 447.514,Z 168.824,A -85,B 0,C 180,E1 -8865.751,E2 -8865.751} C_VEL
LIN {X 0,Y 448.033,Z 157.442,A -85,B 0,C 180,E1 -8868.189,E2 -8868.189} C_VEL
LIN {X 0,Y 447.194,Z 151.688,A -85,B 0,C 180,E1 -8869.492,E2 -8869.492} C_VEL
LIN {X 0,Y 446.523,Z 150.118,A -85,B 0,C 180,E1 -8869.943,E2 -8869.943} C_VEL
LIN {X 0,Y 444.841,Z 148.778,A -85,B 0,C 180,E1 -8870.648,E2 -8870.648} C_VEL
LIN {X 0,Y 442.164,Z 148.406,A -85,B 0,C 180,E1 -8871.615,E2 -8871.615} C_VEL
LIN {X 0,Y 440.408,Z 148.628,A -85,B 0,C 180,E1 -8872.37,E2 -8872.37} C_VEL
LIN {X 0,Y 439.424,Z 148.753,A -85,B 0,C 180,E1 -8873.145,E2 -8873.145} C_VEL
LIN {X 0,Y 439.356,Z 148.756,A -85,B 0,C 180,E1 -8873.407,E2 -8873.407} C_VEL
LIN {X 0,Y 439.369,Z 148.756,A -85,B 0,C 180,E1 -8876.282,E2 -8876.282} C_VEL
LIN {X 0,Y 439.369,Z 148.752,A -85,B 0,C 180,E1 -8879.743,E2 -8879.743} C_VEL
LIN {X 0,Y 439.339,Z 148.762,A -85,B 0,C 180,E1 -8882.36,E2 -8882.36} C_VEL
LIN {X 0,Y 439.385,Z 148.749,A -85,B 0,C 180,E1 -8885.425,E2 -8885.425} C_VEL
LIN {X 0,Y 439.414,Z 148.751,A -85,B 0,C 180,E1 -8888.415,E2 -8888.415} C_VEL
LIN {X 0,Y 439.396,Z 148.748,A -85,B 0,C 180,E1 -8891.343,E2 -8891.343} C_VEL
LIN {X 0,Y 439.42,Z 148.751,A -85,B 0,C 180,E1 -8894.222,E2 -8894.222} C_VEL
LIN {X 0,Y 439.49,Z 148.736,A -85,B 0,C 180,E1 -8897.285,E2 -8897.285} C_VEL
LIN {X 0,Y 439.48,Z 148.737,A -85,B 0,C 180,E1 -8900.797,E2 -8900.797} C_VEL
LIN {X 0,Y 439.563,Z 148.73,A -85,B 0,C 180,E1 -8903.573,E2 -8903.573} C_VEL
LIN {X 0,Y 439.408,Z 148.748,A -85,B 0,C 180,E1 -8905.412,E2 -8905.412} C_VEL
LIN {X 0,Y 439.63,Z 148.722,A -85,B 0,C 180,E1 -8908.167,E2 -8908.167} C_VEL
LIN {X 0,Y 439.673,Z 148.718,A -85,B 0,C 180,E1 -8909.999,E2 -8909.999} C_VEL
LIN {X 0,Y 439.607,Z 148.721,A -85,B 0,C 180,E1 -8912.748,E2 -8912.748} C_VEL
LIN {X 0,Y 439.557,Z 148.728,A -85,B 0,C 180,E1 -8916.425,E2 -8916.425} C_VEL
LIN {X 0,Y 439.478,Z 148.74,A -85,B 0,C 180,E1 -8919.201,E2 -8919.201} C_VEL
LIN {X 0,Y 439.467,Z 148.74,A -85,B 0,C 180,E1 -8922.937,E2 -8922.937} C_VEL
LIN {X 0,Y 439.399,Z 148.747,A -85,B 0,C 180,E1 -8926.325,E2 -8926.325} C_VEL
LIN {X 0,Y 439.378,Z 148.755,A -85,B 0,C 180,E1 -8929.626,E2 -8929.626} C_VEL
LIN {X 0,Y 439.36,Z 148.753,A -85,B 0,C 180,E1 -8932.575,E2 -8932.575} C_VEL
LIN {X 0,Y 439.366,Z 148.755,A -85,B 0,C 180,E1 -8935.586,E2 -8935.586} C_VEL
LIN {X 0,Y 439.38,Z 148.751,A -85,B 0,C 180,E1 -8938.675,E2 -8938.675} C_VEL
LIN {X 0,Y 439.351,Z 148.753,A -85,B 0,C 180,E1 -8942.025,E2 -8942.025} C_VEL
LIN {X 0,Y 439.389,Z 148.753,A -85,B 0,C 180,E1 -8945.338,E2 -8945.338} C_VEL
LIN {X 0,Y 439.365,Z 148.754,A -85,B 0,C 180,E1 -8948.596,E2 -8948.596} C_VEL
LIN {X 0,Y 439.36,Z 148.756,A -85,B 0,C 180,E1 -8951.252,E2 -8951.252} C_VEL
LIN {X 0,Y 439.394,Z 148.754,A -85,B 0,C 180,E1 -8954.729,E2 -8954.729} C_VEL
LIN {X 0,Y 439.345,Z 148.754,A -85,B 0,C 180,E1 -8957.789,E2 -8957.789} C_VEL
LIN {X 0,Y 439.353,Z 148.754,A -85,B 0,C 180,E1 -8961.401,E2 -8961.401} C_VEL
LIN {X 0,Y 439.389,Z 148.754,A -85,B 0,C 180,E1 -8964.843,E2 -8964.843} C_VEL
LIN {X 0,Y 439.361,Z 148.754,A -85,B 0,C 180,E1 -8968.138,E2 -8968.138} C_VEL
LIN {X 0,Y 439.38,Z 148.75,A -85,B 0,C 180,E1 -8971.609,E2 -8971.609} C_VEL
LIN {X 0,Y 439.36,Z 148.759,A -85,B 0,C 180,E1 -8974.412,E2 -8974.412} C_VEL
LIN {X 0,Y 439.353,Z 148.753,A -85,B 0,C 180,E1 -8977.424,E2 -8977.424} C_VEL
LIN {X 0,Y 439.434,Z 148.747,A -85,B 0,C 180,E1 -8980.663,E2 -8980.663} C_VEL
LIN {X 0,Y 439.411,Z 148.753,A -85,B 0,C 180,E1 -8984.222,E2 -8984.222} C_VEL
LIN {X 0,Y 439.477,Z 148.738,A -85,B 0,C 180,E1 -8987.285,E2 -8987.285} C_VEL
LIN {X 0,Y 439.467,Z 148.74,A -85,B 0,C 180,E1 -8990.797,E2 -8990.797} C_VEL
LIN {X 0,Y 439.552,Z 148.73,A -85,B 0,C 180,E1 -8993.574,E2 -8993.574} C_VEL
LIN {X 0,Y 439.397,Z 148.749,A -85,B 0,C 180,E1 -8995.413,E2 -8995.413} C_VEL
LIN {X 0,Y 439.618,Z 148.725,A -85,B 0,C 180,E1 -8998.168,E2 -8998.168} C_VEL
LIN {X 0,Y 439.679,Z 148.719,A -85,B 0,C 180,E1 -9000,E2 -9000} C_VEL
LIN {X 0,Y 439.595,Z 148.723,A -85,B 0,C 180,E1 -9002.749,E2 -9002.749} C_VEL
LIN {X 0,Y 439.549,Z 148.73,A -85,B 0,C 180,E1 -9006.426,E2 -9006.426} C_VEL
LIN {X 0,Y 439.466,Z 148.74,A -85,B 0,C 180,E1 -9009.202,E2 -9009.202} C_VEL
LIN {X 0,Y 439.457,Z 148.741,A -85,B 0,C 180,E1 -9012.938,E2 -9012.938} C_VEL
LIN {X 0,Y 439.389,Z 148.749,A -85,B 0,C 180,E1 -9016.326,E2 -9016.326} C_VEL
LIN {X 0,Y 439.369,Z 148.758,A -85,B 0,C 180,E1 -9019.628,E2 -9019.628} C_VEL
LIN {X 0,Y 439.344,Z 148.754,A -85,B 0,C 180,E1 -9022.576,E2 -9022.576} C_VEL
LIN {X 0,Y 439.358,Z 148.758,A -85,B 0,C 180,E1 -9025.588,E2 -9025.588} C_VEL
LIN {X 0,Y 439.369,Z 148.752,A -85,B 0,C 180,E1 -9028.677,E2 -9028.677} C_VEL
LIN {X 0,Y 439.344,Z 148.755,A -85,B 0,C 180,E1 -9032.027,E2 -9032.027} C_VEL
LIN {X 0,Y 439.38,Z 148.756,A -85,B 0,C 180,E1 -9035.339,E2 -9035.339} C_VEL
LIN {X 0,Y 439.348,Z 148.755,A -85,B 0,C 180,E1 -9038.599,E2 -9038.599} C_VEL
LIN {X 0,Y 439.356,Z 148.758,A -85,B 0,C 180,E1 -9041.253,E2 -9041.253} C_VEL
LIN {X 0,Y 439.39,Z 148.752,A -85,B 0,C 180,E1 -9044.731,E2 -9044.731} C_VEL
LIN {X 0,Y 439.341,Z 148.755,A -85,B 0,C 180,E1 -9047.79,E2 -9047.79} C_VEL
LIN {X 0,Y 439.354,Z 148.754,A -85,B 0,C 180,E1 -9050.221,E2 -9050.221} C_VEL
LIN {X 0,Y 439.361,Z 148.752,A -85,B 0,C 180,E1 -9053.713,E2 -9053.713} C_VEL
LIN {X 0,Y 439.363,Z 148.756,A -85,B 0,C 180,E1 -9057.054,E2 -9057.054} C_VEL
LIN {X 0,Y 439.353,Z 148.757,A -85,B 0,C 180,E1 -9060.273,E2 -9060.273} C_VEL
LIN {X 0,Y 439.379,Z 148.773,A -85,B 0,C 180,E1 -9063.544,E2 -9063.544} C_VEL
LIN {X 0,Y 441.876,Z 162.153,A -85,B 0,C 180,E1 -9066.323,E2 -9066.323} C_VEL
LIN {X 0,Y 441.308,Z 174.828,A -85,B 0,C 180,E1 -9068.759,E2 -9068.759} C_VEL
LIN {X 0,Y 440.473,Z 190.127,A -85,B 0,C 180,E1 -9071.657,E2 -9071.657} C_VEL
LIN {X 0,Y 440.413,Z 191.945,A -85,B 0,C 180,E1 -9072,E2 -9072} C_VEL
LIN {X 0,Y 443.65,Z 213.653,A -85,B 0,C 180,E1 -9072.538,E2 -9072.538} C_VEL
LIN {X 0,Y 442.649,Z 301.051,A -85,B 0,C 180,E1 -9074.106,E2 -9074.106} C_VEL
LIN {X 0,Y 442.204,Z 314.495,A -85,B 0,C 180,E1 -9074.533,E2 -9074.533} C_VEL
LIN {X 0,Y 441.654,Z 327.297,A -85,B 0,C 180,E1 -9075.133,E2 -9075.133} C_VEL
LIN {X 0,Y 441.082,Z 339.852,A -85,B 0,C 180,E1 -9075.938,E2 -9075.938} C_VEL
LIN {X 0,Y 440.52,Z 351.135,A -85,B 0,C 180,E1 -9076.864,E2 -9076.864} C_VEL
LIN {X 0,Y 440.048,Z 360.195,A -85,B 0,C 180,E1 -9077.784,E2 -9077.784} C_VEL
LIN {X 0,Y 439.517,Z 369.528,A -85,B 0,C 180,E1 -9078.938,E2 -9078.938} C_VEL
LIN {X 0,Y 439.024,Z 378.598,A -85,B 0,C 180,E1 -9080.324,E2 -9080.324} C_VEL
LIN {X 0,Y 438.696,Z 385.889,A -85,B 0,C 180,E1 -9081.711,E2 -9081.711} C_VEL
LIN {X 0,Y 438.493,Z 391.685,A -85,B 0,C 180,E1 -9083.097,E2 -9083.097} C_VEL
LIN {X 0,Y 438.372,Z 396.233,A -85,B 0,C 180,E1 -9084.481,E2 -9084.481} C_VEL
LIN {X 0,Y 438.339,Z 398.626,A -85,B 0,C 180,E1 -9085.403,E2 -9085.403} C_VEL
LIN {X 0,Y 438.28,Z 400.577,A -85,B 0,C 180,E1 -9086.323,E2 -9086.323} C_VEL
LIN {X 0,Y 438.34,Z 402.087,A -85,B 0,C 180,E1 -9087.244,E2 -9087.244} C_VEL
LIN {X 0,Y 438.278,Z 403.133,A -85,B 0,C 180,E1 -9088.163,E2 -9088.163} C_VEL
LIN {X 0,Y 438.253,Z 403.78,A -85,B 0,C 180,E1 -9089.082,E2 -9089.082} C_VEL
LIN {X 0,Y 438.255,Z 404.029,A -85,B 0,C 180,E1 -9090.001,E2 -9090.001} C_VEL
LIN {X 0,Y 438.253,Z 403.85,A -85,B 0,C 180,E1 -9090.92,E2 -9090.92} C_VEL
LIN {X 0,Y 438.278,Z 403.24,A -85,B 0,C 180,E1 -9091.839,E2 -9091.839} C_VEL
LIN {X 0,Y 438.34,Z 402.231,A -85,B 0,C 180,E1 -9092.758,E2 -9092.758} C_VEL
LIN {X 0,Y 438.279,Z 400.814,A -85,B 0,C 180,E1 -9093.678,E2 -9093.678} C_VEL
LIN {X 0,Y 438.38,Z 397.828,A -85,B 0,C 180,E1 -9095.059,E2 -9095.059} C_VEL
LIN {X 0,Y 438.448,Z 393.781,A -85,B 0,C 180,E1 -9096.443,E2 -9096.443} C_VEL
LIN {X 0,Y 438.672,Z 387.558,A -85,B 0,C 180,E1 -9098.059,E2 -9098.059} C_VEL
LIN {X 0,Y 439.015,Z 380.751,A -85,B 0,C 180,E1 -9099.445,E2 -9099.445} C_VEL
LIN {X 0,Y 439.438,Z 372.31,A -85,B 0,C 180,E1 -9100.832,E2 -9100.832} C_VEL
LIN {X 0,Y 440.022,Z 363.649,A -85,B 0,C 180,E1 -9101.985,E2 -9101.985} C_VEL
LIN {X 0,Y 440.581,Z 353.968,A -85,B 0,C 180,E1 -9103.042,E2 -9103.042} C_VEL
LIN {X 0,Y 441.198,Z 342.431,A -85,B 0,C 180,E1 -9104.06,E2 -9104.06} C_VEL
LIN {X 0,Y 441.855,Z 330.836,A -85,B 0,C 180,E1 -9104.862,E2 -9104.862} C_VEL
LIN {X 0,Y 442.503,Z 317.61,A -85,B 0,C 180,E1 -9105.547,E2 -9105.547} C_VEL
LIN {X 0,Y 443.025,Z 304.342,A -85,B 0,C 180,E1 -9106.03,E2 -9106.03} C_VEL
LIN {X 0,Y 443.358,Z 288.393,A -85,B 0,C 180,E1 -9106.372,E2 -9106.372} C_VEL
LIN {X 0,Y 444.321,Z 213.619,A -85,B 0,C 180,E1 -9107.734,E2 -9107.734} C_VEL
LIN {X 0,Y 440.877,Z 192.653,A -85,B 0,C 180,E1 -9108.307,E2 -9108.307} C_VEL
LIN {X 0,Y 440.582,Z 190.722,A -85,B 0,C 180,E1 -9108.388,E2 -9108.388} C_VEL
LIN {X 0,Y 441.57,Z 172.89,A -85,B 0,C 180,E1 -9111.719,E2 -9111.719} C_VEL
LIN {X 0,Y 442.037,Z 162.599,A -85,B 0,C 180,E1 -9113.67,E2 -9113.67} C_VEL
LIN {X 0,Y 440.433,Z 153.648,A -85,B 0,C 180,E1 -9115.522,E2 -9115.522} C_VEL
LIN {X 0,Y 439.353,Z 148.762,A -85,B 0,C 180,E1 -9116.609,E2 -9116.609} C_VEL
LIN {X 0,Y 439.359,Z 148.758,A -85,B 0,C 180,E1 -9119.728,E2 -9119.728} C_VEL
LIN {X 0,Y 439.369,Z 148.757,A -85,B 0,C 180,E1 -9122.947,E2 -9122.947} C_VEL
LIN {X 0,Y 439.368,Z 148.754,A -85,B 0,C 180,E1 -9126.289,E2 -9126.289} C_VEL
LIN {X 0,Y 439.361,Z 148.754,A -85,B 0,C 180,E1 -9129.781,E2 -9129.781} C_VEL
LIN {X 0,Y 439.335,Z 148.759,A -85,B 0,C 180,E1 -9132.62,E2 -9132.62} C_VEL
LIN {X 0,Y 439.4,Z 148.748,A -85,B 0,C 180,E1 -9135.271,E2 -9135.271} C_VEL
LIN {X 0,Y 439.356,Z 148.754,A -85,B 0,C 180,E1 -9139.016,E2 -9139.016} C_VEL
LIN {X 0,Y 439.344,Z 148.759,A -85,B 0,C 180,E1 -9142.564,E2 -9142.564} C_VEL
LIN {X 0,Y 439.397,Z 148.754,A -85,B 0,C 180,E1 -9144.844,E2 -9144.844} C_VEL
LIN {X 0,Y 439.372,Z 148.756,A -85,B 0,C 180,E1 -9148.14,E2 -9148.14} C_VEL
LIN {X 0,Y 439.389,Z 148.748,A -85,B 0,C 180,E1 -9151.61,E2 -9151.61} C_VEL
LIN {X 0,Y 439.369,Z 148.754,A -85,B 0,C 180,E1 -9154.413,E2 -9154.413} C_VEL
LIN {X 0,Y 439.365,Z 148.751,A -85,B 0,C 180,E1 -9157.425,E2 -9157.425} C_VEL
LIN {X 0,Y 439.445,Z 148.745,A -85,B 0,C 180,E1 -9160.664,E2 -9160.664} C_VEL
LIN {X 0,Y 439.423,Z 148.75,A -85,B 0,C 180,E1 -9164.223,E2 -9164.223} C_VEL
LIN {X 0,Y 439.489,Z 148.74,A -85,B 0,C 180,E1 -9167.285,E2 -9167.285} C_VEL
LIN {X 0,Y 439.494,Z 148.74,A -85,B 0,C 180,E1 -9170.798,E2 -9170.798} C_VEL
LIN {X 0,Y 439.563,Z 148.734,A -85,B 0,C 180,E1 -9173.574,E2 -9173.574} C_VEL
LIN {X 0,Y 439.412,Z 148.751,A -85,B 0,C 180,E1 -9175.413,E2 -9175.413} C_VEL
LIN {X 0,Y 439.63,Z 148.724,A -85,B 0,C 180,E1 -9178.168,E2 -9178.168} C_VEL
LIN {X 0,Y 439.714,Z 148.717,A -85,B 0,C 180,E1 -9180,E2 -9180} C_VEL
LIN {X 0,Y 439.633,Z 148.726,A -85,B 0,C 180,E1 -9182.749,E2 -9182.749} C_VEL
LIN {X 0,Y 439.596,Z 148.809,A -85,B 0,C 180,E1 -9185.39,E2 -9185.39} C_VEL
LIN {X 0,Y 441.359,Z 158.716,A -85,B 0,C 180,E1 -9187.549,E2 -9187.549} C_VEL
LIN {X 0,Y 441.027,Z 169.434,A -85,B 0,C 180,E1 -9189.71,E2 -9189.71} C_VEL
LIN {X 0,Y 444.622,Z 187.137,A -85,B 0,C 180,E1 -9190.241,E2 -9190.241} C_VEL
LIN {X 0,Y 443.275,Z 278.063,A -85,B 0,C 180,E1 -9191.924,E2 -9191.924} C_VEL
LIN {X 0,Y 442.888,Z 290.963,A -85,B 0,C 180,E1 -9192.341,E2 -9192.341} C_VEL
LIN {X 0,Y 442.471,Z 303.015,A -85,B 0,C 180,E1 -9192.907,E2 -9192.907} C_VEL
LIN {X 0,Y 441.948,Z 315.266,A -85,B 0,C 180,E1 -9193.683,E2 -9193.683} C_VEL
LIN {X 0,Y 441.236,Z 326.995,A -85,B 0,C 180,E1 -9194.636,E2 -9194.636} C_VEL
LIN {X 0,Y 440.579,Z 337.672,A -85,B 0,C 180,E1 -9195.735,E2 -9195.735} C_VEL
LIN {X 0,Y 440.009,Z 347.137,A -85,B 0,C 180,E1 -9196.948,E2 -9196.948} C_VEL
LIN {X 0,Y 439.525,Z 354.924,A -85,B 0,C 180,E1 -9198.168,E2 -9198.168} C_VEL
LIN {X 0,Y 439.202,Z 360.629,A -85,B 0,C 180,E1 -9199.246,E2 -9199.246} C_VEL
LIN {X 0,Y 438.83,Z 366.665,A -85,B 0,C 180,E1 -9200.631,E2 -9200.631} C_VEL
LIN {X 0,Y 438.583,Z 371.754,A -85,B 0,C 180,E1 -9202.121,E2 -9202.121} C_VEL
LIN {X 0,Y 438.419,Z 375.57,A -85,B 0,C 180,E1 -9203.626,E2 -9203.626} C_VEL
LIN {X 0,Y 438.278,Z 377.432,A -85,B 0,C 180,E1 -9204.641,E2 -9204.641} C_VEL
LIN {X 0,Y 438.162,Z 379.209,A -85,B 0,C 180,E1 -9206.073,E2 -9206.073} C_VEL
LIN {X 0,Y 438.134,Z 380.018,A -85,B 0,C 180,E1 -9207.722,E2 -9207.722} C_VEL
LIN {X 0,Y 438.129,Z 379.864,A -85,B 0,C 180,E1 -9208.766,E2 -9208.766} C_VEL
LIN {X 0,Y 438.228,Z 378.974,A -85,B 0,C 180,E1 -9210,E2 -9210} C_VEL
LIN {X 0,Y 438.267,Z 377.913,A -85,B 0,C 180,E1 -9210.874,E2 -9210.874} C_VEL
LIN {X 0,Y 438.374,Z 374.903,A -85,B 0,C 180,E1 -9212.485,E2 -9212.485} C_VEL
LIN {X 0,Y 438.537,Z 370.434,A -85,B 0,C 180,E1 -9214.119,E2 -9214.119} C_VEL
LIN {X 0,Y 438.756,Z 365.428,A -85,B 0,C 180,E1 -9215.497,E2 -9215.497} C_VEL
LIN {X 0,Y 439.051,Z 359.334,A -85,B 0,C 180,E1 -9216.834,E2 -9216.834} C_VEL
LIN {X 0,Y 439.52,Z 351.504,A -85,B 0,C 180,E1 -9218.213,E2 -9218.213} C_VEL
LIN {X 0,Y 440.032,Z 341.963,A -85,B 0,C 180,E1 -9219.559,E2 -9219.559} C_VEL
LIN {X 0,Y 440.546,Z 331.717,A -85,B 0,C 180,E1 -9220.725,E2 -9220.725} C_VEL
LIN {X 0,Y 441.104,Z 321.038,A -85,B 0,C 180,E1 -9221.694,E2 -9221.694} C_VEL
LIN {X 0,Y 441.7,Z 309.147,A -85,B 0,C 180,E1 -9222.55,E2 -9222.55} C_VEL
LIN {X 0,Y 442.138,Z 297.507,A -85,B 0,C 180,E1 -9223.197,E2 -9223.197} C_VEL
LIN {X 0,Y 442.529,Z 283.838,A -85,B 0,C 180,E1 -9223.737,E2 -9223.737} C_VEL
LIN {X 0,Y 442.831,Z 271.148,A -85,B 0,C 180,E1 -9224.054,E2 -9224.054} C_VEL
LIN {X 0,Y 443.829,Z 186.433,A -85,B 0,C 180,E1 -9225.552,E2 -9225.552} C_VEL
LIN {X 0,Y 440.583,Z 168.997,A -85,B 0,C 180,E1 -9226.013,E2 -9226.013} C_VEL
LIN {X 0,Y 441.02,Z 157.546,A -85,B 0,C 180,E1 -9228.503,E2 -9228.503} C_VEL
LIN {X 0,Y 439.375,Z 148.757,A -85,B 0,C 180,E1 -9230.593,E2 -9230.593} C_VEL
LIN {X 0,Y 439.356,Z 148.756,A -85,B 0,C 180,E1 -9233.407,E2 -9233.407} C_VEL
LIN {X 0,Y 438.709,Z 148.839,A -85,B 0,C 180,E1 -9234.173,E2 -9234.173} C_VEL
LIN {X 0,Y 435.832,Z 149.192,A -85,B 0,C 180,E1 -9235.417,E2 -9235.417} C_VEL
LIN {X 0,Y 433.4,Z 149.501,A -85,B 0,C 180,E1 -9236.42,E2 -9236.42} C_VEL
LIN {X 0,Y 432.383,Z 149.622,A -85,B 0,C 180,E1 -9237.197,E2 -9237.197} C_VEL
LIN {X 0,Y 432.315,Z 149.63,A -85,B 0,C 180,E1 -9237.46,E2 -9237.46} C_VEL
LIN {X 0,Y 432.321,Z 149.632,A -85,B 0,C 180,E1 -9240.81,E2 -9240.81} C_VEL
LIN {X 0,Y 432.311,Z 149.633,A -85,B 0,C 180,E1 -9243.963,E2 -9243.963} C_VEL
LIN {X 0,Y 432.307,Z 149.631,A -85,B 0,C 180,E1 -9247.034,E2 -9247.034} C_VEL
LIN {X 0,Y 432.319,Z 149.634,A -85,B 0,C 180,E1 -9250.038,E2 -9250.038} C_VEL
LIN {X 0,Y 432.361,Z 149.625,A -85,B 0,C 180,E1 -9253.547,E2 -9253.547} C_VEL
LIN {X 0,Y 432.436,Z 149.615,A -85,B 0,C 180,E1 -9257.197,E2 -9257.197} C_VEL
LIN {X 0,Y 432.425,Z 149.617,A -85,B 0,C 180,E1 -9260.646,E2 -9260.646} C_VEL
LIN {X 0,Y 432.52,Z 149.606,A -85,B 0,C 180,E1 -9263.468,E2 -9263.468} C_VEL
LIN {X 0,Y 432.377,Z 149.623,A -85,B 0,C 180,E1 -9265.338,E2 -9265.338} C_VEL
LIN {X 0,Y 432.599,Z 149.598,A -85,B 0,C 180,E1 -9268.137,E2 -9268.137} C_VEL
LIN {X 0,Y 432.625,Z 149.596,A -85,B 0,C 180,E1 -9269.999,E2 -9269.999} C_VEL
LIN {X 0,Y 432.561,Z 149.599,A -85,B 0,C 180,E1 -9272.793,E2 -9272.793} C_VEL
LIN {X 0,Y 432.514,Z 149.605,A -85,B 0,C 180,E1 -9276.53,E2 -9276.53} C_VEL
LIN {X 0,Y 432.423,Z 149.62,A -85,B 0,C 180,E1 -9279.353,E2 -9279.353} C_VEL
LIN {X 0,Y 432.433,Z 149.616,A -85,B 0,C 180,E1 -9282.802,E2 -9282.802} C_VEL
LIN {X 0,Y 432.358,Z 149.624,A -85,B 0,C 180,E1 -9286.452,E2 -9286.452} C_VEL
LIN {X 0,Y 432.314,Z 149.631,A -85,B 0,C 180,E1 -9289.961,E2 -9289.961} C_VEL
LIN {X 0,Y 432.309,Z 149.634,A -85,B 0,C 180,E1 -9292.964,E2 -9292.964} C_VEL
LIN {X 0,Y 432.318,Z 149.63,A -85,B 0,C 180,E1 -9296.034,E2 -9296.034} C_VEL
LIN {X 0,Y 432.32,Z 149.637,A -85,B 0,C 180,E1 -9299.188,E2 -9299.188} C_VEL
LIN {X 0,Y 432.315,Z 149.63,A -85,B 0,C 180,E1 -9302.443,E2 -9302.443} C_VEL
LIN {X 0,Y 432.334,Z 149.628,A -85,B 0,C 180,E1 -9305.817,E2 -9305.817} C_VEL
LIN {X 0,Y 432.327,Z 149.632,A -85,B 0,C 180,E1 -9308.711,E2 -9308.711} C_VEL
LIN {X 0,Y 432.3,Z 149.632,A -85,B 0,C 180,E1 -9311.8,E2 -9311.8} C_VEL
LIN {X 0,Y 432.33,Z 149.629,A -85,B 0,C 180,E1 -9314.346,E2 -9314.346} C_VEL
LIN {X 0,Y 432.299,Z 149.637,A -85,B 0,C 180,E1 -9317.017,E2 -9317.017} C_VEL
LIN {X 0,Y 432.284,Z 149.634,A -85,B 0,C 180,E1 -9319.827,E2 -9319.827} C_VEL
LIN {X 0,Y 432.297,Z 149.636,A -85,B 0,C 180,E1 -9323.021,E2 -9323.021} C_VEL
LIN {X 0,Y 432.328,Z 149.629,A -85,B 0,C 180,E1 -9326.001,E2 -9326.001} C_VEL
LIN {X 0,Y 432.335,Z 149.627,A -85,B 0,C 180,E1 -9329.491,E2 -9329.491} C_VEL
LIN {X 0,Y 432.313,Z 149.631,A -85,B 0,C 180,E1 -9331.871,E2 -9331.871} C_VEL
LIN {X 0,Y 432.316,Z 149.631,A -85,B 0,C 180,E1 -9334.996,E2 -9334.996} C_VEL
LIN {X 0,Y 432.348,Z 149.629,A -85,B 0,C 180,E1 -9338.045,E2 -9338.045} C_VEL
LIN {X 0,Y 432.374,Z 149.623,A -85,B 0,C 180,E1 -9341.029,E2 -9341.029} C_VEL
LIN {X 0,Y 432.381,Z 149.625,A -85,B 0,C 180,E1 -9343.959,E2 -9343.959} C_VEL
LIN {X 0,Y 432.447,Z 149.616,A -85,B 0,C 180,E1 -9347.803,E2 -9347.803} C_VEL
LIN {X 0,Y 432.439,Z 149.616,A -85,B 0,C 180,E1 -9351.589,E2 -9351.589} C_VEL
LIN {X 0,Y 432.563,Z 149.602,A -85,B 0,C 180,E1 -9354.405,E2 -9354.405} C_VEL
LIN {X 0,Y 432.587,Z 149.601,A -85,B 0,C 180,E1 -9358.138,E2 -9358.138} C_VEL
LIN {X 0,Y 432.63,Z 149.597,A -85,B 0,C 180,E1 -9360,E2 -9360} C_VEL
LIN {X 0,Y 432.549,Z 149.601,A -85,B 0,C 180,E1 -9362.794,E2 -9362.794} C_VEL
LIN {X 0,Y 432.561,Z 149.604,A -85,B 0,C 180,E1 -9365.594,E2 -9365.594} C_VEL
LIN {X 0,Y 432.438,Z 149.615,A -85,B 0,C 180,E1 -9368.411,E2 -9368.411} C_VEL
LIN {X 0,Y 432.446,Z 149.615,A -85,B 0,C 180,E1 -9372.197,E2 -9372.197} C_VEL
LIN {X 0,Y 432.377,Z 149.625,A -85,B 0,C 180,E1 -9376.041,E2 -9376.041} C_VEL
LIN {X 0,Y 432.339,Z 149.634,A -85,B 0,C 180,E1 -9379.47,E2 -9379.47} C_VEL
LIN {X 0,Y 432.33,Z 149.629,A -85,B 0,C 180,E1 -9382.092,E2 -9382.092} C_VEL
LIN {X 0,Y 432.313,Z 149.633,A -85,B 0,C 180,E1 -9385.003,E2 -9385.003} C_VEL
LIN {X 0,Y 432.306,Z 149.631,A -85,B 0,C 180,E1 -9388.129,E2 -9388.129} C_VEL
LIN {X 0,Y 432.297,Z 149.639,A -85,B 0,C 180,E1 -9391.348,E2 -9391.348} C_VEL
LIN {X 0,Y 432.318,Z 149.631,A -85,B 0,C 180,E1 -9394.679,E2 -9394.679} C_VEL
LIN {X 0,Y 432.315,Z 149.63,A -85,B 0,C 180,E1 -9398.152,E2 -9398.152} C_VEL
LIN {X 0,Y 432.296,Z 149.633,A -85,B 0,C 180,E1 -9401.802,E2 -9401.802} C_VEL
LIN {X 0,Y 432.328,Z 149.629,A -85,B 0,C 180,E1 -9404.348,E2 -9404.348} C_VEL
LIN {X 0,Y 432.295,Z 149.639,A -85,B 0,C 180,E1 -9407.019,E2 -9407.019} C_VEL
LIN {X 0,Y 432.283,Z 149.634,A -85,B 0,C 180,E1 -9409.829,E2 -9409.829} C_VEL
LIN {X 0,Y 432.291,Z 149.638,A -85,B 0,C 180,E1 -9413.022,E2 -9413.022} C_VEL
LIN {X 0,Y 432.328,Z 149.628,A -85,B 0,C 180,E1 -9416.003,E2 -9416.003} C_VEL
LIN {X 0,Y 432.327,Z 149.63,A -85,B 0,C 180,E1 -9419.494,E2 -9419.494} C_VEL
LIN {X 0,Y 432.311,Z 149.632,A -85,B 0,C 180,E1 -9421.873,E2 -9421.873} C_VEL
LIN {X 0,Y 432.331,Z 149.719,A -85,B 0,C 180,E1 -9423.346,E2 -9423.346} C_VEL
LIN {X 0,Y 434.906,Z 163.081,A -85,B 0,C 180,E1 -9426.173,E2 -9426.173} C_VEL
LIN {X 0,Y 434.321,Z 175.769,A -85,B 0,C 180,E1 -9428.65,E2 -9428.65} C_VEL
LIN {X 0,Y 433.516,Z 189.799,A -85,B 0,C 180,E1 -9431.352,E2 -9431.352} C_VEL
LIN {X 0,Y 433.417,Z 191.876,A -85,B 0,C 180,E1 -9431.75,E2 -9431.75} C_VEL
LIN {X 0,Y 436.831,Z 215.53,A -85,B 0,C 180,E1 -9432.324,E2 -9432.324} C_VEL
LIN {X 0,Y 435.763,Z 300.481,A -85,B 0,C 180,E1 -9433.878,E2 -9433.878} C_VEL
LIN {X 0,Y 435.319,Z 314.032,A -85,B 0,C 180,E1 -9434.312,E2 -9434.312} C_VEL
LIN {X 0,Y 434.782,Z 326.405,A -85,B 0,C 180,E1 -9434.892,E2 -9434.892} C_VEL
LIN {X 0,Y 434.135,Z 339.117,A -85,B 0,C 180,E1 -9435.708,E2 -9435.708} C_VEL
LIN {X 0,Y 433.541,Z 350.505,A -85,B 0,C 180,E1 -9436.649,E2 -9436.649} C_VEL
LIN {X 0,Y 433.001,Z 360.684,A -85,B 0,C 180,E1 -9437.701,E2 -9437.701} C_VEL
LIN {X 0,Y 432.38,Z 370.723,A -85,B 0,C 180,E1 -9438.99,E2 -9438.99} C_VEL
LIN {X 0,Y 431.907,Z 379.556,A -85,B 0,C 180,E1 -9440.4,E2 -9440.4} C_VEL
LIN {X 0,Y 431.6,Z 386.583,A -85,B 0,C 180,E1 -9441.809,E2 -9441.809} C_VEL
LIN {X 0,Y 431.375,Z 393.023,A -85,B 0,C 180,E1 -9443.452,E2 -9443.452} C_VEL
LIN {X 0,Y 431.29,Z 397.222,A -85,B 0,C 180,E1 -9444.859,E2 -9444.859} C_VEL
LIN {X 0,Y 431.186,Z 400.325,A -85,B 0,C 180,E1 -9446.263,E2 -9446.263} C_VEL
LIN {X 0,Y 431.236,Z 401.855,A -85,B 0,C 180,E1 -9447.198,E2 -9447.198} C_VEL
LIN {X 0,Y 431.202,Z 402.914,A -85,B 0,C 180,E1 -9448.133,E2 -9448.133} C_VEL
LIN {X 0,Y 431.169,Z 403.57,A -85,B 0,C 180,E1 -9449.067,E2 -9449.067} C_VEL
LIN {X 0,Y 431.169,Z 403.828,A -85,B 0,C 180,E1 -9450.001,E2 -9450.001} C_VEL
LIN {X 0,Y 431.169,Z 403.666,A -85,B 0,C 180,E1 -9450.935,E2 -9450.935} C_VEL
LIN {X 0,Y 431.203,Z 403.063,A -85,B 0,C 180,E1 -9451.869,E2 -9451.869} C_VEL
LIN {X 0,Y 431.235,Z 402.06,A -85,B 0,C 180,E1 -9452.803,E2 -9452.803} C_VEL
LIN {X 0,Y 431.186,Z 400.649,A -85,B 0,C 180,E1 -9453.739,E2 -9453.739} C_VEL
LIN {X 0,Y 431.291,Z 397.674,A -85,B 0,C 180,E1 -9455.143,E2 -9455.143} C_VEL
LIN {X 0,Y 431.377,Z 393.637,A -85,B 0,C 180,E1 -9456.549,E2 -9456.549} C_VEL
LIN {X 0,Y 431.613,Z 387.436,A -85,B 0,C 180,E1 -9458.192,E2 -9458.192} C_VEL
LIN {X 0,Y 431.973,Z 380.649,A -85,B 0,C 180,E1 -9459.6,E2 -9459.6} C_VEL
LIN {X 0,Y 432.454,Z 372.231,A -85,B 0,C 180,E1 -9461.009,E2 -9461.009} C_VEL
LIN {X 0,Y 433.076,Z 363.603,A -85,B 0,C 180,E1 -9462.18,E2 -9462.18} C_VEL
LIN {X 0,Y 433.623,Z 353.344,A -85,B 0,C 180,E1 -9463.316,E2 -9463.316} C_VEL
LIN {X 0,Y 434.321,Z 342.467,A -85,B 0,C 180,E1 -9464.287,E2 -9464.287} C_VEL
LIN {X 0,Y 435.011,Z 330.977,A -85,B 0,C 180,E1 -9465.101,E2 -9465.101} C_VEL
LIN {X 0,Y 435.686,Z 317.9,A -85,B 0,C 180,E1 -9465.796,E2 -9465.796} C_VEL
LIN {X 0,Y 436.243,Z 304.92,A -85,B 0,C 180,E1 -9466.286,E2 -9466.286} C_VEL
LIN {X 0,Y 436.586,Z 291.212,A -85,B 0,C 180,E1 -9466.603,E2 -9466.603} C_VEL
LIN {X 0,Y 437.572,Z 213.833,A -85,B 0,C 180,E1 -9468.049,E2 -9468.049} C_VEL
LIN {X 0,Y 433.979,Z 192.386,A -85,B 0,C 180,E1 -9468.657,E2 -9468.657} C_VEL
LIN {X 0,Y 433.692,Z 190.535,A -85,B 0,C 180,E1 -9468.733,E2 -9468.733} C_VEL
LIN {X 0,Y 434.737,Z 172.92,A -85,B 0,C 180,E1 -9472.078,E2 -9472.078} C_VEL
LIN {X 0,Y 435.125,Z 163.965,A -85,B 0,C 180,E1 -9473.816,E2 -9473.816} C_VEL
LIN {X 0,Y 433.511,Z 155.009,A -85,B 0,C 180,E1 -9475.701,E2 -9475.701} C_VEL
LIN {X 0,Y 432.306,Z 149.641,A -85,B 0,C 180,E1 -9476.9,E2 -9476.9} C_VEL
LIN {X 0,Y 432.317,Z 149.637,A -85,B 0,C 180,E1 -9479.19,E2 -9479.19} C_VEL
LIN {X 0,Y 432.318,Z 149.634,A -85,B 0,C 180,E1 -9482.444,E2 -9482.444} C_VEL
LIN {X 0,Y 432.335,Z 149.631,A -85,B 0,C 180,E1 -9485.819,E2 -9485.819} C_VEL
LIN {X 0,Y 432.302,Z 149.637,A -85,B 0,C 180,E1 -9489.349,E2 -9489.349} C_VEL
LIN {X 0,Y 432.306,Z 149.632,A -85,B 0,C 180,E1 -9491.801,E2 -9491.801} C_VEL
LIN {X 0,Y 432.336,Z 149.628,A -85,B 0,C 180,E1 -9494.348,E2 -9494.348} C_VEL
LIN {X 0,Y 432.305,Z 149.633,A -85,B 0,C 180,E1 -9497.019,E2 -9497.019} C_VEL
LIN {X 0,Y 432.291,Z 149.632,A -85,B 0,C 180,E1 -9499.828,E2 -9499.828} C_VEL
LIN {X 0,Y 432.305,Z 149.633,A -85,B 0,C 180,E1 -9503.022,E2 -9503.022} C_VEL
LIN {X 0,Y 432.336,Z 149.631,A -85,B 0,C 180,E1 -9506.002,E2 -9506.002} C_VEL
LIN {X 0,Y 432.344,Z 149.625,A -85,B 0,C 180,E1 -9509.492,E2 -9509.492} C_VEL
LIN {X 0,Y 432.322,Z 149.63,A -85,B 0,C 180,E1 -9511.873,E2 -9511.873} C_VEL
LIN {X 0,Y 432.327,Z 149.629,A -85,B 0,C 180,E1 -9514.997,E2 -9514.997} C_VEL
LIN {X 0,Y 432.36,Z 149.629,A -85,B 0,C 180,E1 -9518.046,E2 -9518.046} C_VEL
LIN {X 0,Y 432.385,Z 149.622,A -85,B 0,C 180,E1 -9521.03,E2 -9521.03} C_VEL
LIN {X 0,Y 432.392,Z 149.625,A -85,B 0,C 180,E1 -9523.96,E2 -9523.96} C_VEL
LIN {X 0,Y 432.463,Z 149.618,A -85,B 0,C 180,E1 -9527.804,E2 -9527.804} C_VEL
LIN {X 0,Y 432.466,Z 149.619,A -85,B 0,C 180,E1 -9531.59,E2 -9531.59} C_VEL
LIN {X 0,Y 432.576,Z 149.602,A -85,B 0,C 180,E1 -9534.406,E2 -9534.406} C_VEL
LIN {X 0,Y 432.6,Z 149.6,A -85,B 0,C 180,E1 -9538.138,E2 -9538.138} C_VEL
LIN {X 0,Y 432.664,Z 149.595,A -85,B 0,C 180,E1 -9540,E2 -9540} C_VEL
LIN {X 0,Y 432.585,Z 149.604,A -85,B 0,C 180,E1 -9542.794,E2 -9542.794} C_VEL
LIN {X 0,Y 432.471,Z 149.632,A -85,B 0,C 180,E1 -9545.07,E2 -9545.07} C_VEL
LIN {X 0,Y 434.391,Z 159.171,A -85,B 0,C 180,E1 -9547.203,E2 -9547.203} C_VEL
LIN {X 0,Y 434.233,Z 168.589,A -85,B 0,C 180,E1 -9549.146,E2 -9549.146} C_VEL
LIN {X 0,Y 434.2,Z 169.895,A -85,B 0,C 180,E1 -9549.374,E2 -9549.374} C_VEL
LIN {X 0,Y 438,Z 188.093,A -85,B 0,C 180,E1 -9549.933,E2 -9549.933} C_VEL
LIN {X 0,Y 436.52,Z 278.347,A -85,B 0,C 180,E1 -9551.644,E2 -9551.644} C_VEL
LIN {X 0,Y 436.119,Z 291.024,A -85,B 0,C 180,E1 -9552.06,E2 -9552.06} C_VEL
LIN {X 0,Y 435.663,Z 303.185,A -85,B 0,C 180,E1 -9552.638,E2 -9552.638} C_VEL
LIN {X 0,Y 435.124,Z 315.42,A -85,B 0,C 180,E1 -9553.426,E2 -9553.426} C_VEL
LIN {X 0,Y 434.355,Z 327.283,A -85,B 0,C 180,E1 -9554.405,E2 -9554.405} C_VEL
LIN {X 0,Y 433.675,Z 337.837,A -85,B 0,C 180,E1 -9555.51,E2 -9555.51} C_VEL
LIN {X 0,Y 433.052,Z 347.437,A -85,B 0,C 180,E1 -9556.76,E2 -9556.76} C_VEL
LIN {X 0,Y 432.534,Z 355.115,A -85,B 0,C 180,E1 -9557.982,E2 -9557.982} C_VEL
LIN {X 0,Y 432.081,Z 362.216,A -85,B 0,C 180,E1 -9559.368,E2 -9559.368} C_VEL
LIN {X 0,Y 431.687,Z 368.698,A -85,B 0,C 180,E1 -9560.988,E2 -9560.988} C_VEL
LIN {X 0,Y 431.458,Z 373.336,A -85,B 0,C 180,E1 -9562.507,E2 -9562.507} C_VEL
LIN {X 0,Y 431.273,Z 376.933,A -85,B 0,C 180,E1 -9564.135,E2 -9564.135} C_VEL
LIN {X 0,Y 431.144,Z 378.394,A -85,B 0,C 180,E1 -9565.076,E2 -9565.076} C_VEL
LIN {X 0,Y 431.06,Z 379.624,A -85,B 0,C 180,E1 -9566.269,E2 -9566.269} C_VEL
LIN {X 0,Y 431.027,Z 380.127,A -85,B 0,C 180,E1 -9567.165,E2 -9567.165} C_VEL
LIN {X 0,Y 431.03,Z 380.179,A -85,B 0,C 180,E1 -9568.299,E2 -9568.299} C_VEL
LIN {X 0,Y 431.073,Z 379.77,A -85,B 0,C 180,E1 -9569.282,E2 -9569.282} C_VEL
LIN {X 0,Y 431.136,Z 378.783,A -85,B 0,C 180,E1 -9570.354,E2 -9570.354} C_VEL
LIN {X 0,Y 431.258,Z 376.066,A -85,B 0,C 180,E1 -9572.067,E2 -9572.067} C_VEL
LIN {X 0,Y 431.396,Z 372.285,A -85,B 0,C 180,E1 -9573.636,E2 -9573.636} C_VEL
LIN {X 0,Y 431.618,Z 367.406,A -85,B 0,C 180,E1 -9575.127,E2 -9575.127} C_VEL
LIN {X 0,Y 431.946,Z 360.578,A -85,B 0,C 180,E1 -9576.723,E2 -9576.723} C_VEL
LIN {X 0,Y 432.425,Z 352.914,A -85,B 0,C 180,E1 -9578.141,E2 -9578.141} C_VEL
LIN {X 0,Y 432.912,Z 344.264,A -85,B 0,C 180,E1 -9579.433,E2 -9579.433} C_VEL
LIN {X 0,Y 433.396,Z 334.684,A -85,B 0,C 180,E1 -9580.593,E2 -9580.593} C_VEL
LIN {X 0,Y 434.03,Z 323.345,A -85,B 0,C 180,E1 -9581.699,E2 -9581.699} C_VEL
LIN {X 0,Y 434.621,Z 312.81,A -85,B 0,C 180,E1 -9582.515,E2 -9582.515} C_VEL
LIN {X 0,Y 435.139,Z 300.883,A -85,B 0,C 180,E1 -9583.236,E2 -9583.236} C_VEL
LIN {X 0,Y 435.541,Z 287.586,A -85,B 0,C 180,E1 -9583.831,E2 -9583.831} C_VEL
LIN {X 0,Y 435.875,Z 274.197,A -85,B 0,C 180,E1 -9584.216,E2 -9584.216} C_VEL
LIN {X 0,Y 436.955,Z 187.348,A -85,B 0,C 180,E1 -9585.789,E2 -9585.789} C_VEL
LIN {X 0,Y 433.626,Z 169.143,A -85,B 0,C 180,E1 -9586.283,E2 -9586.283} C_VEL
LIN {X 0,Y 434.09,Z 159.486,A -85,B 0,C 180,E1 -9588.409,E2 -9588.409} C_VEL
LIN {X 0,Y 432.34,Z 149.632,A -85,B 0,C 180,E1 -9590.745,E2 -9590.745} C_VEL
LIN {X 0,Y 432.347,Z 149.632,A -85,B 0,C 180,E1 -9594.369,E2 -9594.369} C_VEL
LIN {X 0,Y 432.315,Z 149.63,A -85,B 0,C 180,E1 -9597.46,E2 -9597.46} C_VEL
LIN {X 0,Y 431.697,Z 149.713,A -85,B 0,C 180,E1 -9598.237,E2 -9598.237} C_VEL
LIN {X 0,Y 428.883,Z 150.058,A -85,B 0,C 180,E1 -9599.5,E2 -9599.5} C_VEL
LIN {X 0,Y 426.455,Z 150.366,A -85,B 0,C 180,E1 -9600.52,E2 -9600.52} C_VEL
LIN {X 0,Y 425.379,Z 150.494,A -85,B 0,C 180,E1 -9601.308,E2 -9601.308} C_VEL
LIN {X 0,Y 425.275,Z 150.507,A -85,B 0,C 180,E1 -9601.575,E2 -9601.575} C_VEL
LIN {X 0,Y 425.257,Z 150.514,A -85,B 0,C 180,E1 -9604.551,E2 -9604.551} C_VEL
LIN {X 0,Y 425.295,Z 150.506,A -85,B 0,C 180,E1 -9607.73,E2 -9607.73} C_VEL
LIN {X 0,Y 425.329,Z 150.502,A -85,B 0,C 180,E1 -9610.702,E2 -9610.702} C_VEL
LIN {X 0,Y 425.323,Z 150.503,A -85,B 0,C 180,E1 -9613.685,E2 -9613.685} C_VEL
LIN {X 0,Y 425.398,Z 150.491,A -85,B 0,C 180,E1 -9617.096,E2 -9617.096} C_VEL
LIN {X 0,Y 425.386,Z 150.495,A -85,B 0,C 180,E1 -9620.49,E2 -9620.49} C_VEL
LIN {X 0,Y 425.481,Z 150.482,A -85,B 0,C 180,E1 -9623.36,E2 -9623.36} C_VEL
LIN {X 0,Y 425.347,Z 150.499,A -85,B 0,C 180,E1 -9625.26,E2 -9625.26} C_VEL
LIN {X 0,Y 425.568,Z 150.474,A -85,B 0,C 180,E1 -9628.106,E2 -9628.106} C_VEL
LIN {X 0,Y 425.577,Z 150.474,A -85,B 0,C 180,E1 -9629.999,E2 -9629.999} C_VEL
LIN {X 0,Y 425.516,Z 150.477,A -85,B 0,C 180,E1 -9632.839,E2 -9632.839} C_VEL
LIN {X 0,Y 425.476,Z 150.482,A -85,B 0,C 180,E1 -9636.639,E2 -9636.639} C_VEL
LIN {X 0,Y 425.384,Z 150.499,A -85,B 0,C 180,E1 -9639.509,E2 -9639.509} C_VEL
LIN {X 0,Y 425.396,Z 150.493,A -85,B 0,C 180,E1 -9642.902,E2 -9642.902} C_VEL
LIN {X 0,Y 425.316,Z 150.502,A -85,B 0,C 180,E1 -9646.582,E2 -9646.582} C_VEL
LIN {X 0,Y 425.297,Z 150.509,A -85,B 0,C 180,E1 -9649.622,E2 -9649.622} C_VEL
LIN {X 0,Y 425.287,Z 150.505,A -85,B 0,C 180,E1 -9652.338,E2 -9652.338} C_VEL
LIN {X 0,Y 425.259,Z 150.514,A -85,B 0,C 180,E1 -9655.447,E2 -9655.447} C_VEL
LIN {X 0,Y 425.299,Z 150.507,A -85,B 0,C 180,E1 -9658.857,E2 -9658.857} C_VEL
LIN {X 0,Y 425.252,Z 150.51,A -85,B 0,C 180,E1 -9661.927,E2 -9661.927} C_VEL
LIN {X 0,Y 425.293,Z 150.509,A -85,B 0,C 180,E1 -9665.335,E2 -9665.335} C_VEL
LIN {X 0,Y 425.282,Z 150.512,A -85,B 0,C 180,E1 -9668.899,E2 -9668.899} C_VEL
LIN {X 0,Y 425.262,Z 150.508,A -85,B 0,C 180,E1 -9671.953,E2 -9671.953} C_VEL
LIN {X 0,Y 425.281,Z 150.509,A -85,B 0,C 180,E1 -9675.282,E2 -9675.282} C_VEL
LIN {X 0,Y 425.243,Z 150.516,A -85,B 0,C 180,E1 -9678.617,E2 -9678.617} C_VEL
LIN {X 0,Y 425.273,Z 150.51,A -85,B 0,C 180,E1 -9681.098,E2 -9681.098} C_VEL
LIN {X 0,Y 425.289,Z 150.512,A -85,B 0,C 180,E1 -9684.663,E2 -9684.663} C_VEL
LIN {X 0,Y 425.255,Z 150.511,A -85,B 0,C 180,E1 -9688.072,E2 -9688.072} C_VEL
LIN {X 0,Y 425.289,Z 150.505,A -85,B 0,C 180,E1 -9691.364,E2 -9691.364} C_VEL
LIN {X 0,Y 425.253,Z 150.516,A -85,B 0,C 180,E1 -9694.552,E2 -9694.552} C_VEL
LIN {X 0,Y 425.285,Z 150.506,A -85,B 0,C 180,E1 -9697.729,E2 -9697.729} C_VEL
LIN {X 0,Y 425.353,Z 150.5,A -85,B 0,C 180,E1 -9700.703,E2 -9700.703} C_VEL
LIN {X 0,Y 425.315,Z 150.503,A -85,B 0,C 180,E1 -9703.685,E2 -9703.685} C_VEL
LIN {X 0,Y 425.386,Z 150.493,A -85,B 0,C 180,E1 -9707.097,E2 -9707.097} C_VEL
LIN {X 0,Y 425.373,Z 150.498,A -85,B 0,C 180,E1 -9710.49,E2 -9710.49} C_VEL
LIN {X 0,Y 425.469,Z 150.483,A -85,B 0,C 180,E1 -9713.36,E2 -9713.36} C_VEL
LIN {X 0,Y 425.337,Z 150.499,A -85,B 0,C 180,E1 -9715.261,E2 -9715.261} C_VEL
LIN {X 0,Y 425.556,Z 150.478,A -85,B 0,C 180,E1 -9718.107,E2 -9718.107} C_VEL
LIN {X 0,Y 425.582,Z 150.475,A -85,B 0,C 180,E1 -9720,E2 -9720} C_VEL
LIN {X 0,Y 425.504,Z 150.478,A -85,B 0,C 180,E1 -9722.84,E2 -9722.84} C_VEL
LIN {X 0,Y 425.516,Z 150.482,A -85,B 0,C 180,E1 -9725.687,E2 -9725.687} C_VEL
LIN {X 0,Y 425.386,Z 150.493,A -85,B 0,C 180,E1 -9728.551,E2 -9728.551} C_VEL
LIN {X 0,Y 425.401,Z 150.492,A -85,B 0,C 180,E1 -9732.402,E2 -9732.402} C_VEL
LIN {X 0,Y 425.292,Z 150.508,A -85,B 0,C 180,E1 -9735.331,E2 -9735.331} C_VEL
LIN {X 0,Y 425.275,Z 150.507,A -85,B 0,C 180,E1 -9738.3,E2 -9738.3} C_VEL
LIN {X 0,Y 425.272,Z 150.512,A -85,B 0,C 180,E1 -9741.319,E2 -9741.319} C_VEL
LIN {X 0,Y 425.287,Z 150.506,A -85,B 0,C 180,E1 -9744.65,E2 -9744.65} C_VEL
LIN {X 0,Y 425.235,Z 150.517,A -85,B 0,C 180,E1 -9747.566,E2 -9747.566} C_VEL
LIN {X 0,Y 425.277,Z 150.508,A -85,B 0,C 180,E1 -9750.76,E2 -9750.76} C_VEL
LIN {X 0,Y 425.283,Z 150.506,A -85,B 0,C 180,E1 -9754.284,E2 -9754.284} C_VEL
LIN {X 0,Y 425.263,Z 150.51,A -85,B 0,C 180,E1 -9757.696,E2 -9757.696} C_VEL
LIN {X 0,Y 425.236,Z 150.513,A -85,B 0,C 180,E1 -9760.515,E2 -9760.515} C_VEL
LIN {X 0,Y 425.238,Z 150.515,A -85,B 0,C 180,E1 -9763.35,E2 -9763.35} C_VEL
LIN {X 0,Y 425.25,Z 150.51,A -85,B 0,C 180,E1 -9766.044,E2 -9766.044} C_VEL
LIN {X 0,Y 425.242,Z 150.514,A -85,B 0,C 180,E1 -9768.619,E2 -9768.619} C_VEL
LIN {X 0,Y 425.271,Z 150.512,A -85,B 0,C 180,E1 -9771.1,E2 -9771.1} C_VEL
LIN {X 0,Y 425.288,Z 150.511,A -85,B 0,C 180,E1 -9774.664,E2 -9774.664} C_VEL
LIN {X 0,Y 425.248,Z 150.511,A -85,B 0,C 180,E1 -9778.073,E2 -9778.073} C_VEL
LIN {X 0,Y 425.288,Z 150.508,A -85,B 0,C 180,E1 -9781.366,E2 -9781.366} C_VEL
LIN {X 0,Y 425.288,Z 150.614,A -85,B 0,C 180,E1 -9783.138,E2 -9783.138} C_VEL
LIN {X 0,Y 427.913,Z 163.995,A -85,B 0,C 180,E1 -9786.016,E2 -9786.016} C_VEL
LIN {X 0,Y 427.579,Z 174.156,A -85,B 0,C 180,E1 -9788.042,E2 -9788.042} C_VEL
LIN {X 0,Y 426.452,Z 191.539,A -85,B 0,C 180,E1 -9791.442,E2 -9791.442} C_VEL
LIN {X 0,Y 426.485,Z 192.059,A -85,B 0,C 180,E1 -9791.489,E2 -9791.489} C_VEL
LIN {X 0,Y 429.986,Z 215.11,A -85,B 0,C 180,E1 -9792.064,E2 -9792.064} C_VEL
LIN {X 0,Y 428.862,Z 300.962,A -85,B 0,C 180,E1 -9793.672,E2 -9793.672} C_VEL
LIN {X 0,Y 428.398,Z 314.282,A -85,B 0,C 180,E1 -9794.113,E2 -9794.113} C_VEL
LIN {X 0,Y 427.839,Z 326.52,A -85,B 0,C 180,E1 -9794.702,E2 -9794.702} C_VEL
LIN {X 0,Y 427.195,Z 338.363,A -85,B 0,C 180,E1 -9795.471,E2 -9795.471} C_VEL
LIN {X 0,Y 426.629,Z 349.467,A -85,B 0,C 180,E1 -9796.392,E2 -9796.392} C_VEL
LIN {X 0,Y 425.947,Z 360.146,A -85,B 0,C 180,E1 -9797.494,E2 -9797.494} C_VEL
LIN {X 0,Y 425.384,Z 370.257,A -85,B 0,C 180,E1 -9798.807,E2 -9798.807} C_VEL
LIN {X 0,Y 424.876,Z 379.151,A -85,B 0,C 180,E1 -9800.239,E2 -9800.239} C_VEL
LIN {X 0,Y 424.532,Z 386.228,A -85,B 0,C 180,E1 -9801.672,E2 -9801.672} C_VEL
LIN {X 0,Y 424.298,Z 392.705,A -85,B 0,C 180,E1 -9803.343,E2 -9803.343} C_VEL
LIN {X 0,Y 424.202,Z 396.936,A -85,B 0,C 180,E1 -9804.773,E2 -9804.773} C_VEL
LIN {X 0,Y 424.098,Z 400.068,A -85,B 0,C 180,E1 -9806.2,E2 -9806.2} C_VEL
LIN {X 0,Y 424.132,Z 401.616,A -85,B 0,C 180,E1 -9807.151,E2 -9807.151} C_VEL
LIN {X 0,Y 424.128,Z 402.693,A -85,B 0,C 180,E1 -9808.102,E2 -9808.102} C_VEL
LIN {X 0,Y 424.089,Z 403.359,A -85,B 0,C 180,E1 -9809.051,E2 -9809.051} C_VEL
LIN {X 0,Y 424.086,Z 403.626,A -85,B 0,C 180,E1 -9810.001,E2 -9810.001} C_VEL
LIN {X 0,Y 424.089,Z 403.481,A -85,B 0,C 180,E1 -9810.95,E2 -9810.95} C_VEL
LIN {X 0,Y 424.129,Z 402.888,A -85,B 0,C 180,E1 -9811.9,E2 -9811.9} C_VEL
LIN {X 0,Y 424.13,Z 401.892,A -85,B 0,C 180,E1 -9812.85,E2 -9812.85} C_VEL
LIN {X 0,Y 424.097,Z 400.489,A -85,B 0,C 180,E1 -9813.802,E2 -9813.802} C_VEL
LIN {X 0,Y 424.203,Z 397.53,A -85,B 0,C 180,E1 -9815.229,E2 -9815.229} C_VEL
LIN {X 0,Y 424.301,Z 393.511,A -85,B 0,C 180,E1 -9816.659,E2 -9816.659} C_VEL
LIN {X 0,Y 424.569,Z 387.333,A -85,B 0,C 180,E1 -9818.329,E2 -9818.329} C_VEL
LIN {X 0,Y 424.945,Z 380.561,A -85,B 0,C 180,E1 -9819.761,E2 -9819.761} C_VEL
LIN {X 0,Y 425.45,Z 372.171,A -85,B 0,C 180,E1 -9821.193,E2 -9821.193} C_VEL
LIN {X 0,Y 426.133,Z 363.588,A -85,B 0,C 180,E1 -9822.381,E2 -9822.381} C_VEL
LIN {X 0,Y 426.736,Z 352.881,A -85,B 0,C 180,E1 -9823.586,E2 -9823.586} C_VEL
LIN {X 0,Y 427.535,Z 341.113,A -85,B 0,C 180,E1 -9824.641,E2 -9824.641} C_VEL
LIN {X 0,Y 428.309,Z 329.218,A -85,B 0,C 180,E1 -9825.465,E2 -9825.465} C_VEL
LIN {X 0,Y 429.015,Z 315.713,A -85,B 0,C 180,E1 -9826.171,E2 -9826.171} C_VEL
LIN {X 0,Y 429.534,Z 303.718,A -85,B 0,C 180,E1 -9826.609,E2 -9826.609} C_VEL
LIN {X 0,Y 429.898,Z 287.869,A -85,B 0,C 180,E1 -9826.961,E2 -9826.961} C_VEL
LIN {X 0,Y 430.937,Z 214.854,A -85,B 0,C 180,E1 -9828.356,E2 -9828.356} C_VEL
LIN {X 0,Y 427.354,Z 193.401,A -85,B 0,C 180,E1 -9828.986,E2 -9828.986} C_VEL
LIN {X 0,Y 426.795,Z 190.256,A -85,B 0,C 180,E1 -9829.11,E2 -9829.11} C_VEL
LIN {X 0,Y 427.905,Z 173.1,A -85,B 0,C 180,E1 -9832.434,E2 -9832.434} C_VEL
LIN {X 0,Y 428.222,Z 165.331,A -85,B 0,C 180,E1 -9833.967,E2 -9833.967} C_VEL
LIN {X 0,Y 426.589,Z 156.432,A -85,B 0,C 180,E1 -9835.887,E2 -9835.887} C_VEL
LIN {X 0,Y 425.259,Z 150.518,A -85,B 0,C 180,E1 -9837.256,E2 -9837.256} C_VEL
LIN {X 0,Y 425.273,Z 150.512,A -85,B 0,C 180,E1 -9839.722,E2 -9839.722} C_VEL
LIN {X 0,Y 425.269,Z 150.515,A -85,B 0,C 180,E1 -9843.05,E2 -9843.05} C_VEL
LIN {X 0,Y 425.279,Z 150.509,A -85,B 0,C 180,E1 -9845.928,E2 -9845.928} C_VEL
LIN {X 0,Y 425.261,Z 150.515,A -85,B 0,C 180,E1 -9849.037,E2 -9849.037} C_VEL
LIN {X 0,Y 425.259,Z 150.512,A -85,B 0,C 180,E1 -9852.656,E2 -9852.656} C_VEL
LIN {X 0,Y 425.288,Z 150.506,A -85,B 0,C 180,E1 -9855.284,E2 -9855.284} C_VEL
LIN {X 0,Y 425.25,Z 150.51,A -85,B 0,C 180,E1 -9858.618,E2 -9858.618} C_VEL
LIN {X 0,Y 425.281,Z 150.505,A -85,B 0,C 180,E1 -9861.099,E2 -9861.099} C_VEL
LIN {X 0,Y 425.297,Z 150.509,A -85,B 0,C 180,E1 -9864.664,E2 -9864.664} C_VEL
LIN {X 0,Y 425.265,Z 150.512,A -85,B 0,C 180,E1 -9868.073,E2 -9868.073} C_VEL
LIN {X 0,Y 425.298,Z 150.503,A -85,B 0,C 180,E1 -9871.365,E2 -9871.365} C_VEL
LIN {X 0,Y 425.263,Z 150.511,A -85,B 0,C 180,E1 -9874.553,E2 -9874.553} C_VEL
LIN {X 0,Y 425.295,Z 150.505,A -85,B 0,C 180,E1 -9877.73,E2 -9877.73} C_VEL
LIN {X 0,Y 425.364,Z 150.498,A -85,B 0,C 180,E1 -9880.704,E2 -9880.704} C_VEL
LIN {X 0,Y 425.326,Z 150.506,A -85,B 0,C 180,E1 -9883.686,E2 -9883.686} C_VEL
LIN {X 0,Y 425.398,Z 150.495,A -85,B 0,C 180,E1 -9887.097,E2 -9887.097} C_VEL
LIN {X 0,Y 425.398,Z 150.497,A -85,B 0,C 180,E1 -9890.491,E2 -9890.491} C_VEL
LIN {X 0,Y 425.48,Z 150.488,A -85,B 0,C 180,E1 -9893.361,E2 -9893.361} C_VEL
LIN {X 0,Y 425.351,Z 150.502,A -85,B 0,C 180,E1 -9895.261,E2 -9895.261} C_VEL
LIN {X 0,Y 425.569,Z 150.476,A -85,B 0,C 180,E1 -9898.107,E2 -9898.107} C_VEL
LIN {X 0,Y 425.615,Z 150.473,A -85,B 0,C 180,E1 -9900,E2 -9900} C_VEL
LIN {X 0,Y 425.539,Z 150.482,A -85,B 0,C 180,E1 -9902.84,E2 -9902.84} C_VEL
LIN {X 0,Y 425.366,Z 150.541,A -85,B 0,C 180,E1 -9904.739,E2 -9904.739} C_VEL
LIN {X 0,Y 427.14,Z 158.666,A -85,B 0,C 180,E1 -9906.614,E2 -9906.614} C_VEL
LIN {X 0,Y 427.641,Z 162.958,A -85,B 0,C 180,E1 -9907.555,E2 -9907.555} C_VEL
LIN {X 0,Y 427.359,Z 169.794,A -85,B 0,C 180,E1 -9908.979,E2 -9908.979} C_VEL
LIN {X 0,Y 431.326,Z 188.678,A -85,B 0,C 180,E1 -9909.604,E2 -9909.604} C_VEL
LIN {X 0,Y 429.812,Z 278.539,A -85,B 0,C 180,E1 -9911.346,E2 -9911.346} C_VEL
LIN {X 0,Y 429.39,Z 291.359,A -85,B 0,C 180,E1 -9911.776,E2 -9911.776} C_VEL
LIN {X 0,Y 428.882,Z 303.432,A -85,B 0,C 180,E1 -9912.36,E2 -9912.36} C_VEL
LIN {X 0,Y 428.299,Z 315.643,A -85,B 0,C 180,E1 -9913.161,E2 -9913.161} C_VEL
LIN {X 0,Y 427.558,Z 326.992,A -85,B 0,C 180,E1 -9914.111,E2 -9914.111} C_VEL
LIN {X 0,Y 426.865,Z 336.985,A -85,B 0,C 180,E1 -9915.152,E2 -9915.152} C_VEL
LIN {X 0,Y 426.21,Z 346.793,A -85,B 0,C 180,E1 -9916.424,E2 -9916.424} C_VEL
LIN {X 0,Y 425.562,Z 355.32,A -85,B 0,C 180,E1 -9917.79,E2 -9917.79} C_VEL
LIN {X 0,Y 425.024,Z 362.924,A -85,B 0,C 180,E1 -9919.312,E2 -9919.312} C_VEL
LIN {X 0,Y 424.642,Z 368.903,A -85,B 0,C 180,E1 -9920.845,E2 -9920.845} C_VEL
LIN {X 0,Y 424.386,Z 373.545,A -85,B 0,C 180,E1 -9922.389,E2 -9922.389} C_VEL
LIN {X 0,Y 424.261,Z 375.974,A -85,B 0,C 180,E1 -9923.426,E2 -9923.426} C_VEL
LIN {X 0,Y 424.145,Z 377.83,A -85,B 0,C 180,E1 -9924.472,E2 -9924.472} C_VEL
LIN {X 0,Y 424.007,Z 379.222,A -85,B 0,C 180,E1 -9925.529,E2 -9925.529} C_VEL
LIN {X 0,Y 423.942,Z 380.071,A -85,B 0,C 180,E1 -9926.59,E2 -9926.59} C_VEL
LIN {X 0,Y 423.927,Z 380.416,A -85,B 0,C 180,E1 -9927.658,E2 -9927.658} C_VEL
LIN {X 0,Y 423.955,Z 380.256,A -85,B 0,C 180,E1 -9928.734,E2 -9928.734} C_VEL
LIN {X 0,Y 424.059,Z 378.832,A -85,B 0,C 180,E1 -9930.479,E2 -9930.479} C_VEL
LIN {X 0,Y 424.188,Z 375.814,A -85,B 0,C 180,E1 -9932.33,E2 -9932.33} C_VEL
LIN {X 0,Y 424.315,Z 372.677,A -85,B 0,C 180,E1 -9933.618,E2 -9933.618} C_VEL
LIN {X 0,Y 424.595,Z 366.842,A -85,B 0,C 180,E1 -9935.404,E2 -9935.404} C_VEL
LIN {X 0,Y 424.942,Z 359.852,A -85,B 0,C 180,E1 -9937.02,E2 -9937.02} C_VEL
LIN {X 0,Y 425.408,Z 353.025,A -85,B 0,C 180,E1 -9938.282,E2 -9938.282} C_VEL
LIN {X 0,Y 425.881,Z 344.826,A -85,B 0,C 180,E1 -9939.53,E2 -9939.53} C_VEL
LIN {X 0,Y 426.363,Z 335.495,A -85,B 0,C 180,E1 -9940.689,E2 -9940.689} C_VEL
LIN {X 0,Y 427.01,Z 324.385,A -85,B 0,C 180,E1 -9941.804,E2 -9941.804} C_VEL
LIN {X 0,Y 427.708,Z 312.345,A -85,B 0,C 180,E1 -9942.753,E2 -9942.753} C_VEL
LIN {X 0,Y 428.256,Z 300.157,A -85,B 0,C 180,E1 -9943.49,E2 -9943.49} C_VEL
LIN {X 0,Y 428.663,Z 286.849,A -85,B 0,C 180,E1 -9944.081,E2 -9944.081} C_VEL
LIN {X 0,Y 429.037,Z 273.392,A -85,B 0,C 180,E1 -9944.458,E2 -9944.458} C_VEL
LIN {X 0,Y 430.19,Z 188.565,A -85,B 0,C 180,E1 -9946.025,E2 -9946.025} C_VEL
LIN {X 0,Y 426.68,Z 169.4,A -85,B 0,C 180,E1 -9946.538,E2 -9946.538} C_VEL
LIN {X 0,Y 427.082,Z 160.273,A -85,B 0,C 180,E1 -9948.577,E2 -9948.577} C_VEL
LIN {X 0,Y 425.288,Z 150.511,A -85,B 0,C 180,E1 -9950.959,E2 -9950.959} C_VEL
LIN {X 0,Y 425.285,Z 150.511,A -85,B 0,C 180,E1 -9954.072,E2 -9954.072} C_VEL
LIN {X 0,Y 425.279,Z 150.506,A -85,B 0,C 180,E1 -9957.45,E2 -9957.45} C_VEL
LIN {X 0,Y 425.277,Z 150.512,A -85,B 0,C 180,E1 -9960.279,E2 -9960.279} C_VEL
LIN {X 0,Y 425.275,Z 150.507,A -85,B 0,C 180,E1 -9961.575,E2 -9961.575} C_VEL
LIN {X 0,Y 424.566,Z 150.602,A -85,B 0,C 180,E1 -9962.365,E2 -9962.365} C_VEL
LIN {X 0,Y 421.708,Z 150.952,A -85,B 0,C 180,E1 -9963.65,E2 -9963.65} C_VEL
LIN {X 0,Y 419.324,Z 151.251,A -85,B 0,C 180,E1 -9964.687,E2 -9964.687} C_VEL
LIN {X 0,Y 418.314,Z 151.375,A -85,B 0,C 180,E1 -9965.488,E2 -9965.488} C_VEL
LIN {X 0,Y 418.237,Z 151.385,A -85,B 0,C 180,E1 -9965.759,E2 -9965.759} C_VEL
LIN {X 0,Y 418.231,Z 151.391,A -85,B 0,C 180,E1 -9968.303,E2 -9968.303} C_VEL
LIN {X 0,Y 418.243,Z 151.383,A -85,B 0,C 180,E1 -9971.38,E2 -9971.38} C_VEL
LIN {X 0,Y 418.253,Z 151.386,A -85,B 0,C 180,E1 -9974.403,E2 -9974.403} C_VEL
LIN {X 0,Y 418.359,Z 151.369,A -85,B 0,C 180,E1 -9977.385,E2 -9977.385} C_VEL
LIN {X 0,Y 418.372,Z 151.367,A -85,B 0,C 180,E1 -9981.304,E2 -9981.304} C_VEL
LIN {X 0,Y 418.474,Z 151.358,A -85,B 0,C 180,E1 -9984.216,E2 -9984.216} C_VEL
LIN {X 0,Y 418.537,Z 151.351,A -85,B 0,C 180,E1 -9988.075,E2 -9988.075} C_VEL
LIN {X 0,Y 418.41,Z 151.362,A -85,B 0,C 180,E1 -9990.962,E2 -9990.962} C_VEL
LIN {X 0,Y 418.473,Z 151.354,A -85,B 0,C 180,E1 -9992.887,E2 -9992.887} C_VEL
LIN {X 0,Y 418.441,Z 151.358,A -85,B 0,C 180,E1 -9996.751,E2 -9996.751} C_VEL
LIN {X 0,Y 418.324,Z 151.379,A -85,B 0,C 180,E1 -9999.671,E2 -9999.671} C_VEL
LIN {X 0,Y 418.349,Z 151.371,A -85,B 0,C 180,E1 -10002.999,E2 -10002.999} C_VEL
LIN {X 0,Y 418.259,Z 151.381,A -85,B 0,C 180,E1 -10006.709,E2 -10006.709} C_VEL
LIN {X 0,Y 418.243,Z 151.386,A -85,B 0,C 180,E1 -10009.778,E2 -10009.778} C_VEL
LIN {X 0,Y 418.227,Z 151.386,A -85,B 0,C 180,E1 -10012.736,E2 -10012.736} C_VEL
LIN {X 0,Y 418.218,Z 151.387,A -85,B 0,C 180,E1 -10015.906,E2 -10015.906} C_VEL
LIN {X 0,Y 418.256,Z 151.388,A -85,B 0,C 180,E1 -10019.162,E2 -10019.162} C_VEL
LIN {X 0,Y 418.247,Z 151.386,A -85,B 0,C 180,E1 -10022.841,E2 -10022.841} C_VEL
LIN {X 0,Y 418.241,Z 151.383,A -85,B 0,C 180,E1 -10026.236,E2 -10026.236} C_VEL
LIN {X 0,Y 418.207,Z 151.388,A -85,B 0,C 180,E1 -10029.686,E2 -10029.686} C_VEL
LIN {X 0,Y 418.205,Z 151.389,A -85,B 0,C 180,E1 -10032.317,E2 -10032.317} C_VEL
LIN {X 0,Y 418.232,Z 151.388,A -85,B 0,C 180,E1 -10035.108,E2 -10035.108} C_VEL
LIN {X 0,Y 418.215,Z 151.386,A -85,B 0,C 180,E1 -10037.763,E2 -10037.763} C_VEL
LIN {X 0,Y 418.231,Z 151.384,A -85,B 0,C 180,E1 -10041.555,E2 -10041.555} C_VEL
LIN {X 0,Y 418.245,Z 151.384,A -85,B 0,C 180,E1 -10045.157,E2 -10045.157} C_VEL
LIN {X 0,Y 418.237,Z 151.384,A -85,B 0,C 180,E1 -10047.471,E2 -10047.471} C_VEL
LIN {X 0,Y 418.253,Z 151.385,A -85,B 0,C 180,E1 -10050.897,E2 -10050.897} C_VEL
LIN {X 0,Y 418.212,Z 151.389,A -85,B 0,C 180,E1 -10054.092,E2 -10054.092} C_VEL
LIN {X 0,Y 418.22,Z 151.386,A -85,B 0,C 180,E1 -10057.262,E2 -10057.262} C_VEL
LIN {X 0,Y 418.276,Z 151.386,A -85,B 0,C 180,E1 -10060.363,E2 -10060.363} C_VEL
LIN {X 0,Y 418.272,Z 151.379,A -85,B 0,C 180,E1 -10063.402,E2 -10063.402} C_VEL
LIN {X 0,Y 418.339,Z 151.371,A -85,B 0,C 180,E1 -10067,E2 -10067} C_VEL
LIN {X 0,Y 418.314,Z 151.379,A -85,B 0,C 180,E1 -10070.328,E2 -10070.328} C_VEL
LIN {X 0,Y 418.434,Z 151.359,A -85,B 0,C 180,E1 -10073.248,E2 -10073.248} C_VEL
LIN {X 0,Y 418.309,Z 151.375,A -85,B 0,C 180,E1 -10075.181,E2 -10075.181} C_VEL
LIN {X 0,Y 418.525,Z 151.354,A -85,B 0,C 180,E1 -10078.075,E2 -10078.075} C_VEL
LIN {X 0,Y 418.534,Z 151.353,A -85,B 0,C 180,E1 -10080,E2 -10080} C_VEL
LIN {X 0,Y 418.461,Z 151.356,A -85,B 0,C 180,E1 -10082.888,E2 -10082.888} C_VEL
LIN {X 0,Y 418.474,Z 151.361,A -85,B 0,C 180,E1 -10085.783,E2 -10085.783} C_VEL
LIN {X 0,Y 418.359,Z 151.368,A -85,B 0,C 180,E1 -10088.696,E2 -10088.696} C_VEL
LIN {X 0,Y 418.345,Z 151.37,A -85,B 0,C 180,E1 -10092.615,E2 -10092.615} C_VEL
LIN {X 0,Y 418.241,Z 151.39,A -85,B 0,C 180,E1 -10095.596,E2 -10095.596} C_VEL
LIN {X 0,Y 418.229,Z 151.384,A -85,B 0,C 180,E1 -10098.619,E2 -10098.619} C_VEL
LIN {X 0,Y 418.218,Z 151.391,A -85,B 0,C 180,E1 -10101.697,E2 -10101.697} C_VEL
LIN {X 0,Y 418.236,Z 151.385,A -85,B 0,C 180,E1 -10104.853,E2 -10104.853} C_VEL
LIN {X 0,Y 418.195,Z 151.389,A -85,B 0,C 180,E1 -10108.07,E2 -10108.07} C_VEL
LIN {X 0,Y 418.227,Z 151.389,A -85,B 0,C 180,E1 -10111.019,E2 -10111.019} C_VEL
LIN {X 0,Y 418.224,Z 151.387,A -85,B 0,C 180,E1 -10113.679,E2 -10113.679} C_VEL
LIN {X 0,Y 418.226,Z 151.392,A -85,B 0,C 180,E1 -10117.226,E2 -10117.226} C_VEL
LIN {X 0,Y 418.2,Z 151.393,A -85,B 0,C 180,E1 -10120.868,E2 -10120.868} C_VEL
LIN {X 0,Y 418.195,Z 151.389,A -85,B 0,C 180,E1 -10123.729,E2 -10123.729} C_VEL
LIN {X 0,Y 418.193,Z 151.391,A -85,B 0,C 180,E1 -10126.448,E2 -10126.448} C_VEL
LIN {X 0,Y 418.201,Z 151.393,A -85,B 0,C 180,E1 -10129.134,E2 -10129.134} C_VEL
LIN {X 0,Y 418.228,Z 151.391,A -85,B 0,C 180,E1 -10132.776,E2 -10132.776} C_VEL
LIN {X 0,Y 418.227,Z 151.387,A -85,B 0,C 180,E1 -10136.322,E2 -10136.322} C_VEL
LIN {X 0,Y 418.23,Z 151.386,A -85,B 0,C 180,E1 -10139.728,E2 -10139.728} C_VEL
LIN {X 0,Y 418.245,Z 151.548,A -85,B 0,C 180,E1 -10142.932,E2 -10142.932} C_VEL
LIN {X 0,Y 420.896,Z 164.89,A -85,B 0,C 180,E1 -10145.853,E2 -10145.853} C_VEL
LIN {X 0,Y 420.785,Z 170.74,A -85,B 0,C 180,E1 -10147.046,E2 -10147.046} C_VEL
LIN {X 0,Y 419.921,Z 185.458,A -85,B 0,C 180,E1 -10149.992,E2 -10149.992} C_VEL
LIN {X 0,Y 419.477,Z 191.599,A -85,B 0,C 180,E1 -10151.201,E2 -10151.201} C_VEL
LIN {X 0,Y 423.145,Z 216.529,A -85,B 0,C 180,E1 -10151.838,E2 -10151.838} C_VEL
LIN {X 0,Y 421.985,Z 300.166,A -85,B 0,C 180,E1 -10153.429,E2 -10153.429} C_VEL
LIN {X 0,Y 421.466,Z 313.652,A -85,B 0,C 180,E1 -10153.875,E2 -10153.875} C_VEL
LIN {X 0,Y 420.913,Z 326.542,A -85,B 0,C 180,E1 -10154.506,E2 -10154.506} C_VEL
LIN {X 0,Y 420.183,Z 339.129,A -85,B 0,C 180,E1 -10155.347,E2 -10155.347} C_VEL
LIN {X 0,Y 419.586,Z 350.102,A -85,B 0,C 180,E1 -10156.286,E2 -10156.286} C_VEL
LIN {X 0,Y 418.899,Z 360.559,A -85,B 0,C 180,E1 -10157.403,E2 -10157.403} C_VEL
LIN {X 0,Y 418.389,Z 369.748,A -85,B 0,C 180,E1 -10158.617,E2 -10158.617} C_VEL
LIN {X 0,Y 417.853,Z 378.708,A -85,B 0,C 180,E1 -10160.074,E2 -10160.074} C_VEL
LIN {X 0,Y 417.49,Z 385.852,A -85,B 0,C 180,E1 -10161.531,E2 -10161.531} C_VEL
LIN {X 0,Y 417.23,Z 392.37,A -85,B 0,C 180,E1 -10163.229,E2 -10163.229} C_VEL
LIN {X 0,Y 417.116,Z 396.637,A -85,B 0,C 180,E1 -10164.684,E2 -10164.684} C_VEL
LIN {X 0,Y 417.013,Z 399.801,A -85,B 0,C 180,E1 -10166.135,E2 -10166.135} C_VEL
LIN {X 0,Y 417.029,Z 401.368,A -85,B 0,C 180,E1 -10167.103,E2 -10167.103} C_VEL
LIN {X 0,Y 417.056,Z 402.467,A -85,B 0,C 180,E1 -10168.069,E2 -10168.069} C_VEL
LIN {X 0,Y 417.011,Z 403.145,A -85,B 0,C 180,E1 -10169.035,E2 -10169.035} C_VEL
LIN {X 0,Y 417.005,Z 403.423,A -85,B 0,C 180,E1 -10170.001,E2 -10170.001} C_VEL
LIN {X 0,Y 417.011,Z 403.295,A -85,B 0,C 180,E1 -10170.966,E2 -10170.966} C_VEL
LIN {X 0,Y 417.056,Z 402.716,A -85,B 0,C 180,E1 -10171.932,E2 -10171.932} C_VEL
LIN {X 0,Y 417.027,Z 401.728,A -85,B 0,C 180,E1 -10172.899,E2 -10172.899} C_VEL
LIN {X 0,Y 417.013,Z 400.333,A -85,B 0,C 180,E1 -10173.866,E2 -10173.866} C_VEL
LIN {X 0,Y 417.117,Z 397.391,A -85,B 0,C 180,E1 -10175.318,E2 -10175.318} C_VEL
LIN {X 0,Y 417.234,Z 393.393,A -85,B 0,C 180,E1 -10176.772,E2 -10176.772} C_VEL
LIN {X 0,Y 417.511,Z 387.249,A -85,B 0,C 180,E1 -10178.471,E2 -10178.471} C_VEL
LIN {X 0,Y 417.913,Z 380.502,A -85,B 0,C 180,E1 -10179.927,E2 -10179.927} C_VEL
LIN {X 0,Y 418.468,Z 372.132,A -85,B 0,C 180,E1 -10181.382,E2 -10181.382} C_VEL
LIN {X 0,Y 419.195,Z 363.594,A -85,B 0,C 180,E1 -10182.589,E2 -10182.589} C_VEL
LIN {X 0,Y 419.751,Z 353.896,A -85,B 0,C 180,E1 -10183.718,E2 -10183.718} C_VEL
